TYPE "udt_API_Login"
VERSION : 0.1
   STRUCT
      Username : String[128];   // Username as entered in the login window / Request
      Password : String[128];   // User password as entered in the login window / Request
      AutoLogoffTime : Int;   // Minutes after the client must perform the logout if the user is idle.  / Response
      UserGroup : String[128];   // Name of the user group that the user belongs to. / Response
      LoginTriggerAndResponse : Int;   // 0 = ready/idle; 1 = request; 2 = OK (Login successful); 10 = UserNotFound; 11 = WrongPassword; 12 = Disabled; 13 = Locked; 14 = PasswordChangeRequired; 15 = PasswordChangeRequiredDomainUser / TriggerAndResponse
   END_STRUCT;

END_TYPE

TYPE "udt_API_Logout"
VERSION : 0.1
   STRUCT
      LogoutTriggerAndResponse : Int;   // 0 = ready/idle; 1 = request; 2 = OK (logout successful) / TriggerAndResponse
   END_STRUCT;

END_TYPE

TYPE "udt_API_Authorization"
VERSION : 0.1
   STRUCT
      AccessRightCustomId : String[20];   // Custom Id of the access right that the authorization is carried out against. / Request
      AuthorizationTriggerAndResponse : Int;   // 0 = ready/idle; 1 = request; 2 = OK (Authorized); 3 = OK (NotAuthorized); 4 = OK (Challenged): 12 = NoUserIsLoggedIn; 13 = AccessRightNotFound / TriggerAndResponse
      ElectronicSignatureType : Int;   // 0 = cleared; 1 = Confirmation only, optional comment; 2 = Confirmation only, required comment; 3 = Authenticated signature, optional comment; 4 = Authenticated signature, required comment / Response (optional)
      ElectronicSignatureName : String[128];   // Name of the required electronic signature / Response (optional)
      ElectronicSignatureUsername : String[128];   // Username to sign the electronic signature / Request (optional)
      ElectronicSignaturePassword : String[128];   // Password to sign the electronic signature / Request (optional)
      ElecronicSignatureComment : String[128];   // Comment provided with signing of the signature / Request (optional)
      ElectronicSignatureChallengeStatus : Int;   // 0 = cleared; 2 = OK; 10 = SignatoryAuthenticationError; 11 = SignatoryNotAuthorized; 12 = CommentRequired / Response (optional)
   END_STRUCT;

END_TYPE

TYPE "udt_API_UserDefinedEvent"
VERSION : 0.1
   STRUCT
      EventCustomId : String[20];   // Custom Id of the user defined event that is logged to the audit trail. / Request
      EventData : String[200];   // Data associated with the event (string separated with #).  / Request
      UserDefinedEventTriggerAndResponse : Int;   // 0 = ready/idle; 1 = request; 2 = OK (Event successfully written); 10 = EventCustomIdNotFound; 11 = EventDataNotConsistentWithEventTemplate / TriggerAndResponse
   END_STRUCT;

END_TYPE

TYPE "udt_API_StepRecipeDownload"
VERSION : 0.1
   STRUCT
      RecipeId : DInt;   // Id of selected recipe / Request
      StepNumber : DInt;   // Step number of the operation to be downloaded. First step starts with 1 / Request
      OperationId : DInt;   // Id of the operation that must be executed for the current procedural element.  / Response
      CreatedFromProceduralElement : DInt;   // Id of the procedural element, which is used to display the report data on the report. API writes the id of the procedural element from the recipe.  / Response
      StepRecipeDownloadTriggerAndResponse : Int;   // 0 = ready/idle; 1 = request; 2 = OK (step downloaded); 3 = OK (end of recipe); 10 = RecipeIdNotFound; 11 = ParameterAddressNotFoundOnServer; 12 = NonLinearRecipe; 13 = RecipeContainsNoSteps; 14 = NegativeOrZeroStepNumber; 15 = RecipeDoesNotHaveStepNumber / TriggerAndResponse
   END_STRUCT;

END_TYPE

TYPE "udt_API_TimeSync"
VERSION : 0.1
   STRUCT
      TimeSyncTriggerAndResponse : Int;   // 0 = ready/idle; 1 = request; 2 = OK (Time data sent) / TriggerAndResponse
      CurrentUnixServerTime : DInt;   // UNIX timestamp (seconds since Jan 01, 1970. (UTC)) / Response
      CurrentLocalServerTime : Date_And_Time;   // Current local server time in date time format. / Response
      CurrentUtcServerTime : Date_And_Time;   // Current UTC server time in date time format. / Response
      CurrentServerTimeOffset : Int;   // Number of hours representing the time offset from UTC / Response
   END_STRUCT;

END_TYPE

TYPE "udt_API_Watchdog"
VERSION : 0.1
   STRUCT
      IsApiResponsive : Bool;   // Periodically set to true by the API. Client should reset to false before checking the status of the service.  / Response
   END_STRUCT;

END_TYPE

TYPE "udt_API_ReportHeaderCreate"
VERSION : 0.1
   STRUCT
      StartUser : String[128];   // Name of the user that executed actions resulting in the generation of the report. / Request
      RecipeId : DInt;   // Id of the recipe that was executed to generate the report (in recipe regime only). Leave value at 0 for non-recipe regime. / Request (Optional)
      BatchId : DInt;   // Id of the batch that was executed to generate the report (in recipe regime only, if batches are used). Leave value at 0 if batch is not used. / Response
      ReportHeaderId : DInt;   // Id of the created report header. / Response
      ReportHeaderCreateTriggerAndResponse : Int;   // 0 = ready/idle; 1 = request; 2 = OK (Report header created); 10 = RecipeIdNotFound; 11 = BatchIdNotFound; 12 = RecipeIsNotLocalRecipe / TriggerAndResponse
   END_STRUCT;

END_TYPE

TYPE "udt_API_ReportStepUpload"
VERSION : 0.1
   STRUCT
      ReportHeaderId : DInt;   // Id of the report header to which the procedural element will be added. / Request
      OperationId : DInt;   // Id of the operation whose parameters are uploaded to the database. / Request
      StartDate : Date_And_Time;   // Start date and time of the procedural element / Request
      EndDate : Date_And_Time;   // End date and time of the procedural element / Request
      ExecutionStatus : Int;   // 0 = successful; 1 = failed; 2 = aborted / Request
      CreatedFromProceduralElement : DInt;   // Id of the procedural element from which the report data is created / Request (optional)
      ReportStepUploadTriggerAndResponse : Int;   // 0 = ready/idle; 1 = request; 2 = OK (Report step uploaded); 10 = ReportHeaderIdNotFound; 11 = OperationIdNotFound; 12 = InvalidExecutionStatus; 13 = ParameterAddressNotFoundOnServer; 14 = StartDateAfterEndDate / TriggerAndResponse
   END_STRUCT;

END_TYPE

TYPE "udt_API_ReportFinish"
VERSION : 0.1
   STRUCT
      EndUser : String[128];   // Name of the user that executed actions resulting in the completion of the report.
      ReportHeaderId : DInt;   // Id of the report header to be concluded
      ReportFinishTriggerAndResponse : Int;   // 0 = ready/idle, 1 = request, 2 = OK (Report header concluded), 10 = ReportHeaderIdNotFound
   END_STRUCT;

END_TYPE

TYPE "udt_API_Full"
VERSION : 0.1
   STRUCT
      Login : "udt_API_Login";
      Logout : "udt_API_Logout";
      Authorization : "udt_API_Authorization";
      UserDefinedEvent : "udt_API_UserDefinedEvent";
      StepRecipeDownload : "udt_API_StepRecipeDownload";
      TimeSync : "udt_API_TimeSync";
      Watchdog : "udt_API_Watchdog";
      ReportHeaderCreate : "udt_API_ReportHeaderCreate";
      ReportStepUpload : "udt_API_ReportStepUpload";
      ReportFinish : "udt_API_ReportFinish";
   END_STRUCT;

END_TYPE

TYPE "udtUnit"
VERSION : 0.1
   STRUCT
      Regime : Int;   //  Control mode (0=automatic, 1=manual, 2=service)
      Status : Int;   //  Unit status
      ID : Int;   //  Unit ID
      Ready : Int;   //  0 = Ready; 1 = not ready
      Enable : Bool;   //  1-Unit is Enabled
      Alocated : Bool;   //  1-Unit is alocated
      Spare1 : Bool;   // spare
      Active : Bool;   //  1-Unit is active
      AlarmAck : Bool;   //  1 = Akcknowledge all unit alarms
      interaction : Bool;   //  1 = unit request for operator interaction
      PhaseH : Bool;   //  1 = one or more phases are HELD
      PhaseF : Bool;   //  1 = one or more phases are in alarm
      Simulation : Bool;   // Enable Simulation on SCADA (ifix)
      Spare2 : Bool;   // Enable Simulation on HMI (siemens panel)
      Spare3 : Bool;   // spare
      Spare4 : Bool;
      Spare5 : Bool;
      Spare6 : Bool;
      Spare7 : Bool;
      Spare8 : Bool;
   END_STRUCT;

END_TYPE

DATA_BLOCK "dbAPI"
{ S7_Optimized_Access := 'FALSE' }
VERSION : 0.1
NON_RETAIN
   STRUCT
      PdbmApi : Array[0..4] of "udt_API_Full";
   END_STRUCT;


BEGIN
   PdbmApi[0].Login.Username := '';
   PdbmApi[0].Login.Password := '';
   PdbmApi[0].Login.AutoLogoffTime := 0;
   PdbmApi[0].Login.UserGroup := '';
   PdbmApi[0].Login.LoginTriggerAndResponse := 0;
   PdbmApi[0].Logout.LogoutTriggerAndResponse := 0;
   PdbmApi[0].Authorization.AccessRightCustomId := '';
   PdbmApi[0].Authorization.AuthorizationTriggerAndResponse := 0;
   PdbmApi[0].Authorization.ElectronicSignatureType := 0;
   PdbmApi[0].Authorization.ElectronicSignatureName := '';
   PdbmApi[0].Authorization.ElectronicSignatureUsername := '';
   PdbmApi[0].Authorization.ElectronicSignaturePassword := '';
   PdbmApi[0].Authorization.ElecronicSignatureComment := '';
   PdbmApi[0].Authorization.ElectronicSignatureChallengeStatus := 0;
   PdbmApi[0].UserDefinedEvent.EventCustomId := '';
   PdbmApi[0].UserDefinedEvent.EventData := '';
   PdbmApi[0].UserDefinedEvent.UserDefinedEventTriggerAndResponse := 2;
   PdbmApi[0].StepRecipeDownload.RecipeId := 0;
   PdbmApi[0].StepRecipeDownload.StepNumber := 0;
   PdbmApi[0].StepRecipeDownload.OperationId := 95;
   PdbmApi[0].StepRecipeDownload.CreatedFromProceduralElement := 157;
   PdbmApi[0].StepRecipeDownload.StepRecipeDownloadTriggerAndResponse := 0;
   PdbmApi[0].TimeSync.TimeSyncTriggerAndResponse := 0;
   PdbmApi[0].TimeSync.CurrentUnixServerTime := 1_671_231_209;
   PdbmApi[0].TimeSync.CurrentLocalServerTime := DT#2022-12-17-00:53:29.655;
   PdbmApi[0].TimeSync.CurrentUtcServerTime := DT#2022-12-16-22:53:29.656;
   PdbmApi[0].TimeSync.CurrentServerTimeOffset := 2;
   PdbmApi[0].Watchdog.IsApiResponsive := FALSE;
   PdbmApi[0].ReportHeaderCreate.StartUser := '';
   PdbmApi[0].ReportHeaderCreate.RecipeId := 0;
   PdbmApi[0].ReportHeaderCreate.BatchId := 0;
   PdbmApi[0].ReportHeaderCreate.ReportHeaderId := 1491;
   PdbmApi[0].ReportHeaderCreate.ReportHeaderCreateTriggerAndResponse := 0;
   PdbmApi[0].ReportStepUpload.ReportHeaderId := 0;
   PdbmApi[0].ReportStepUpload.OperationId := 0;
   PdbmApi[0].ReportStepUpload.StartDate := DT#1990-01-01-00:00:00;
   PdbmApi[0].ReportStepUpload.EndDate := DT#1990-01-01-00:00:00;
   PdbmApi[0].ReportStepUpload.ExecutionStatus := 0;
   PdbmApi[0].ReportStepUpload.CreatedFromProceduralElement := 0;
   PdbmApi[0].ReportStepUpload.ReportStepUploadTriggerAndResponse := 0;
   PdbmApi[0].ReportFinish.EndUser := '';
   PdbmApi[0].ReportFinish.ReportHeaderId := 0;
   PdbmApi[0].ReportFinish.ReportFinishTriggerAndResponse := 2;
   PdbmApi[1].Login.Username := '';
   PdbmApi[1].Login.Password := '';
   PdbmApi[1].Login.AutoLogoffTime := 60;
   PdbmApi[1].Login.UserGroup := 'ADMINISTRATOR';
   PdbmApi[1].Login.LoginTriggerAndResponse := 0;
   PdbmApi[1].Logout.LogoutTriggerAndResponse := 2;
   PdbmApi[1].Authorization.AccessRightCustomId := '';
   PdbmApi[1].Authorization.AuthorizationTriggerAndResponse := 0;
   PdbmApi[1].Authorization.ElectronicSignatureType := 0;
   PdbmApi[1].Authorization.ElectronicSignatureName := '';
   PdbmApi[1].Authorization.ElectronicSignatureUsername := '';
   PdbmApi[1].Authorization.ElectronicSignaturePassword := '';
   PdbmApi[1].Authorization.ElecronicSignatureComment := '';
   PdbmApi[1].Authorization.ElectronicSignatureChallengeStatus := 0;
   PdbmApi[1].UserDefinedEvent.EventCustomId := '';
   PdbmApi[1].UserDefinedEvent.EventData := '';
   PdbmApi[1].UserDefinedEvent.UserDefinedEventTriggerAndResponse := 2;
   PdbmApi[1].StepRecipeDownload.RecipeId := 0;
   PdbmApi[1].StepRecipeDownload.StepNumber := 0;
   PdbmApi[1].StepRecipeDownload.OperationId := 0;
   PdbmApi[1].StepRecipeDownload.CreatedFromProceduralElement := 0;
   PdbmApi[1].StepRecipeDownload.StepRecipeDownloadTriggerAndResponse := 0;
   PdbmApi[1].TimeSync.TimeSyncTriggerAndResponse := 0;
   PdbmApi[1].TimeSync.CurrentUnixServerTime := 0;
   PdbmApi[1].TimeSync.CurrentLocalServerTime := DT#1990-01-01-00:00:00;
   PdbmApi[1].TimeSync.CurrentUtcServerTime := DT#1990-01-01-00:00:00;
   PdbmApi[1].TimeSync.CurrentServerTimeOffset := 0;
   PdbmApi[1].Watchdog.IsApiResponsive := TRUE;
   PdbmApi[1].ReportHeaderCreate.StartUser := '';
   PdbmApi[1].ReportHeaderCreate.RecipeId := 0;
   PdbmApi[1].ReportHeaderCreate.BatchId := 0;
   PdbmApi[1].ReportHeaderCreate.ReportHeaderId := 0;
   PdbmApi[1].ReportHeaderCreate.ReportHeaderCreateTriggerAndResponse := 0;
   PdbmApi[1].ReportStepUpload.ReportHeaderId := 0;
   PdbmApi[1].ReportStepUpload.OperationId := 0;
   PdbmApi[1].ReportStepUpload.StartDate := DT#1990-01-01-00:00:00;
   PdbmApi[1].ReportStepUpload.EndDate := DT#1990-01-01-00:00:00;
   PdbmApi[1].ReportStepUpload.ExecutionStatus := 0;
   PdbmApi[1].ReportStepUpload.CreatedFromProceduralElement := 0;
   PdbmApi[1].ReportStepUpload.ReportStepUploadTriggerAndResponse := 0;
   PdbmApi[1].ReportFinish.EndUser := '';
   PdbmApi[1].ReportFinish.ReportHeaderId := 0;
   PdbmApi[1].ReportFinish.ReportFinishTriggerAndResponse := 0;
   PdbmApi[2].Login.Username := '';
   PdbmApi[2].Login.Password := '';
   PdbmApi[2].Login.AutoLogoffTime := 60;
   PdbmApi[2].Login.UserGroup := 'ADMINISTRATOR';
   PdbmApi[2].Login.LoginTriggerAndResponse := 0;
   PdbmApi[2].Logout.LogoutTriggerAndResponse := 2;
   PdbmApi[2].Authorization.AccessRightCustomId := '0';
   PdbmApi[2].Authorization.AuthorizationTriggerAndResponse := 0;
   PdbmApi[2].Authorization.ElectronicSignatureType := 0;
   PdbmApi[2].Authorization.ElectronicSignatureName := '';
   PdbmApi[2].Authorization.ElectronicSignatureUsername := '';
   PdbmApi[2].Authorization.ElectronicSignaturePassword := '';
   PdbmApi[2].Authorization.ElecronicSignatureComment := '';
   PdbmApi[2].Authorization.ElectronicSignatureChallengeStatus := 0;
   PdbmApi[2].UserDefinedEvent.EventCustomId := '';
   PdbmApi[2].UserDefinedEvent.EventData := '';
   PdbmApi[2].UserDefinedEvent.UserDefinedEventTriggerAndResponse := 2;
   PdbmApi[2].StepRecipeDownload.RecipeId := 0;
   PdbmApi[2].StepRecipeDownload.StepNumber := 0;
   PdbmApi[2].StepRecipeDownload.OperationId := 0;
   PdbmApi[2].StepRecipeDownload.CreatedFromProceduralElement := 0;
   PdbmApi[2].StepRecipeDownload.StepRecipeDownloadTriggerAndResponse := 0;
   PdbmApi[2].TimeSync.TimeSyncTriggerAndResponse := 0;
   PdbmApi[2].TimeSync.CurrentUnixServerTime := 0;
   PdbmApi[2].TimeSync.CurrentLocalServerTime := DT#1990-01-01-00:00:00;
   PdbmApi[2].TimeSync.CurrentUtcServerTime := DT#1990-01-01-00:00:00;
   PdbmApi[2].TimeSync.CurrentServerTimeOffset := 0;
   PdbmApi[2].Watchdog.IsApiResponsive := TRUE;
   PdbmApi[2].ReportHeaderCreate.StartUser := '';
   PdbmApi[2].ReportHeaderCreate.RecipeId := 0;
   PdbmApi[2].ReportHeaderCreate.BatchId := 0;
   PdbmApi[2].ReportHeaderCreate.ReportHeaderId := 0;
   PdbmApi[2].ReportHeaderCreate.ReportHeaderCreateTriggerAndResponse := 0;
   PdbmApi[2].ReportStepUpload.ReportHeaderId := 0;
   PdbmApi[2].ReportStepUpload.OperationId := 0;
   PdbmApi[2].ReportStepUpload.StartDate := DT#1990-01-01-00:00:00;
   PdbmApi[2].ReportStepUpload.EndDate := DT#1990-01-01-00:00:00;
   PdbmApi[2].ReportStepUpload.ExecutionStatus := 0;
   PdbmApi[2].ReportStepUpload.CreatedFromProceduralElement := 0;
   PdbmApi[2].ReportStepUpload.ReportStepUploadTriggerAndResponse := 0;
   PdbmApi[2].ReportFinish.EndUser := '';
   PdbmApi[2].ReportFinish.ReportHeaderId := 0;
   PdbmApi[2].ReportFinish.ReportFinishTriggerAndResponse := 0;
   PdbmApi[3].Login.Username := '';
   PdbmApi[3].Login.Password := '';
   PdbmApi[3].Login.AutoLogoffTime := 60;
   PdbmApi[3].Login.UserGroup := 'ADMINISTRATOR';
   PdbmApi[3].Login.LoginTriggerAndResponse := 0;
   PdbmApi[3].Logout.LogoutTriggerAndResponse := 2;
   PdbmApi[3].Authorization.AccessRightCustomId := '';
   PdbmApi[3].Authorization.AuthorizationTriggerAndResponse := 0;
   PdbmApi[3].Authorization.ElectronicSignatureType := 0;
   PdbmApi[3].Authorization.ElectronicSignatureName := '';
   PdbmApi[3].Authorization.ElectronicSignatureUsername := '';
   PdbmApi[3].Authorization.ElectronicSignaturePassword := '';
   PdbmApi[3].Authorization.ElecronicSignatureComment := '';
   PdbmApi[3].Authorization.ElectronicSignatureChallengeStatus := 0;
   PdbmApi[3].UserDefinedEvent.EventCustomId := '';
   PdbmApi[3].UserDefinedEvent.EventData := '';
   PdbmApi[3].UserDefinedEvent.UserDefinedEventTriggerAndResponse := 2;
   PdbmApi[3].StepRecipeDownload.RecipeId := 0;
   PdbmApi[3].StepRecipeDownload.StepNumber := 0;
   PdbmApi[3].StepRecipeDownload.OperationId := 0;
   PdbmApi[3].StepRecipeDownload.CreatedFromProceduralElement := 0;
   PdbmApi[3].StepRecipeDownload.StepRecipeDownloadTriggerAndResponse := 0;
   PdbmApi[3].TimeSync.TimeSyncTriggerAndResponse := 0;
   PdbmApi[3].TimeSync.CurrentUnixServerTime := 0;
   PdbmApi[3].TimeSync.CurrentLocalServerTime := DT#1990-01-01-00:00:00;
   PdbmApi[3].TimeSync.CurrentUtcServerTime := DT#1990-01-01-00:00:00;
   PdbmApi[3].TimeSync.CurrentServerTimeOffset := 0;
   PdbmApi[3].Watchdog.IsApiResponsive := TRUE;
   PdbmApi[3].ReportHeaderCreate.StartUser := '';
   PdbmApi[3].ReportHeaderCreate.RecipeId := 0;
   PdbmApi[3].ReportHeaderCreate.BatchId := 0;
   PdbmApi[3].ReportHeaderCreate.ReportHeaderId := 0;
   PdbmApi[3].ReportHeaderCreate.ReportHeaderCreateTriggerAndResponse := 0;
   PdbmApi[3].ReportStepUpload.ReportHeaderId := 0;
   PdbmApi[3].ReportStepUpload.OperationId := 0;
   PdbmApi[3].ReportStepUpload.StartDate := DT#1990-01-01-00:00:00;
   PdbmApi[3].ReportStepUpload.EndDate := DT#1990-01-01-00:00:00;
   PdbmApi[3].ReportStepUpload.ExecutionStatus := 0;
   PdbmApi[3].ReportStepUpload.CreatedFromProceduralElement := 0;
   PdbmApi[3].ReportStepUpload.ReportStepUploadTriggerAndResponse := 0;
   PdbmApi[3].ReportFinish.EndUser := '';
   PdbmApi[3].ReportFinish.ReportHeaderId := 0;
   PdbmApi[3].ReportFinish.ReportFinishTriggerAndResponse := 0;
   PdbmApi[4].Login.Username := '';
   PdbmApi[4].Login.Password := '';
   PdbmApi[4].Login.AutoLogoffTime := 0;
   PdbmApi[4].Login.UserGroup := '';
   PdbmApi[4].Login.LoginTriggerAndResponse := 0;
   PdbmApi[4].Logout.LogoutTriggerAndResponse := 0;
   PdbmApi[4].Authorization.AccessRightCustomId := '';
   PdbmApi[4].Authorization.AuthorizationTriggerAndResponse := 0;
   PdbmApi[4].Authorization.ElectronicSignatureType := 0;
   PdbmApi[4].Authorization.ElectronicSignatureName := '';
   PdbmApi[4].Authorization.ElectronicSignatureUsername := '';
   PdbmApi[4].Authorization.ElectronicSignaturePassword := '';
   PdbmApi[4].Authorization.ElecronicSignatureComment := '';
   PdbmApi[4].Authorization.ElectronicSignatureChallengeStatus := 0;
   PdbmApi[4].UserDefinedEvent.EventCustomId := '';
   PdbmApi[4].UserDefinedEvent.EventData := '';
   PdbmApi[4].UserDefinedEvent.UserDefinedEventTriggerAndResponse := 0;
   PdbmApi[4].StepRecipeDownload.RecipeId := 0;
   PdbmApi[4].StepRecipeDownload.StepNumber := 0;
   PdbmApi[4].StepRecipeDownload.OperationId := 0;
   PdbmApi[4].StepRecipeDownload.CreatedFromProceduralElement := 0;
   PdbmApi[4].StepRecipeDownload.StepRecipeDownloadTriggerAndResponse := 0;
   PdbmApi[4].TimeSync.TimeSyncTriggerAndResponse := 0;
   PdbmApi[4].TimeSync.CurrentUnixServerTime := 0;
   PdbmApi[4].TimeSync.CurrentLocalServerTime := DT#1990-01-01-00:00:00;
   PdbmApi[4].TimeSync.CurrentUtcServerTime := DT#1990-01-01-00:00:00;
   PdbmApi[4].TimeSync.CurrentServerTimeOffset := 0;
   PdbmApi[4].Watchdog.IsApiResponsive := TRUE;
   PdbmApi[4].ReportHeaderCreate.StartUser := '';
   PdbmApi[4].ReportHeaderCreate.RecipeId := 0;
   PdbmApi[4].ReportHeaderCreate.BatchId := 0;
   PdbmApi[4].ReportHeaderCreate.ReportHeaderId := 145;
   PdbmApi[4].ReportHeaderCreate.ReportHeaderCreateTriggerAndResponse := 2;
   PdbmApi[4].ReportStepUpload.ReportHeaderId := 0;
   PdbmApi[4].ReportStepUpload.OperationId := 0;
   PdbmApi[4].ReportStepUpload.StartDate := DT#1990-01-01-00:00:00;
   PdbmApi[4].ReportStepUpload.EndDate := DT#1990-01-01-00:00:00;
   PdbmApi[4].ReportStepUpload.ExecutionStatus := 0;
   PdbmApi[4].ReportStepUpload.CreatedFromProceduralElement := 0;
   PdbmApi[4].ReportStepUpload.ReportStepUploadTriggerAndResponse := 2;
   PdbmApi[4].ReportFinish.EndUser := '';
   PdbmApi[4].ReportFinish.ReportHeaderId := 0;
   PdbmApi[4].ReportFinish.ReportFinishTriggerAndResponse := 0;

END_DATA_BLOCK

DATA_BLOCK "dbUnit"
{ S7_Optimized_Access := 'FALSE' }
VERSION : 0.1
   STRUCT
      Unit : Array[1..10] of "udtUnit";
   END_STRUCT;


BEGIN
   Unit[1].Regime := 0;
   Unit[1].Status := 2;
   Unit[1].ID := 1;
   Unit[1].Ready := 0;
   Unit[1].Enable := TRUE;
   Unit[1].Alocated := FALSE;
   Unit[1].Spare1 := FALSE;
   Unit[1].Active := TRUE;
   Unit[1].AlarmAck := FALSE;
   Unit[1].interaction := FALSE;
   Unit[1].PhaseH := TRUE;
   Unit[1].PhaseF := FALSE;
   Unit[1].Simulation := TRUE;
   Unit[1].Spare2 := FALSE;
   Unit[1].Spare3 := FALSE;
   Unit[1].Spare4 := FALSE;
   Unit[1].Spare5 := FALSE;
   Unit[1].Spare6 := FALSE;
   Unit[1].Spare7 := FALSE;
   Unit[1].Spare8 := FALSE;
   Unit[2].Regime := 0;
   Unit[2].Status := 2;
   Unit[2].ID := 2;
   Unit[2].Ready := 0;
   Unit[2].Enable := TRUE;
   Unit[2].Alocated := FALSE;
   Unit[2].Spare1 := FALSE;
   Unit[2].Active := TRUE;
   Unit[2].AlarmAck := TRUE;
   Unit[2].interaction := FALSE;
   Unit[2].PhaseH := TRUE;
   Unit[2].PhaseF := FALSE;
   Unit[2].Simulation := FALSE;
   Unit[2].Spare2 := FALSE;
   Unit[2].Spare3 := FALSE;
   Unit[2].Spare4 := FALSE;
   Unit[2].Spare5 := FALSE;
   Unit[2].Spare6 := FALSE;
   Unit[2].Spare7 := FALSE;
   Unit[2].Spare8 := FALSE;
   Unit[3].Regime := 0;
   Unit[3].Status := 2;
   Unit[3].ID := 3;
   Unit[3].Ready := 0;
   Unit[3].Enable := TRUE;
   Unit[3].Alocated := FALSE;
   Unit[3].Spare1 := FALSE;
   Unit[3].Active := TRUE;
   Unit[3].AlarmAck := TRUE;
   Unit[3].interaction := TRUE;
   Unit[3].PhaseH := FALSE;
   Unit[3].PhaseF := FALSE;
   Unit[3].Simulation := FALSE;
   Unit[3].Spare2 := FALSE;
   Unit[3].Spare3 := FALSE;
   Unit[3].Spare4 := FALSE;
   Unit[3].Spare5 := FALSE;
   Unit[3].Spare6 := FALSE;
   Unit[3].Spare7 := FALSE;
   Unit[3].Spare8 := FALSE;
   Unit[4].Regime := 0;
   Unit[4].Status := 2;
   Unit[4].ID := 4;
   Unit[4].Ready := 0;
   Unit[4].Enable := TRUE;
   Unit[4].Alocated := FALSE;
   Unit[4].Spare1 := FALSE;
   Unit[4].Active := TRUE;
   Unit[4].AlarmAck := TRUE;
   Unit[4].interaction := FALSE;
   Unit[4].PhaseH := TRUE;
   Unit[4].PhaseF := FALSE;
   Unit[4].Simulation := FALSE;
   Unit[4].Spare2 := FALSE;
   Unit[4].Spare3 := FALSE;
   Unit[4].Spare4 := FALSE;
   Unit[4].Spare5 := FALSE;
   Unit[4].Spare6 := FALSE;
   Unit[4].Spare7 := FALSE;
   Unit[4].Spare8 := FALSE;
   Unit[5].Regime := 0;
   Unit[5].Status := 2;
   Unit[5].ID := 5;
   Unit[5].Ready := 0;
   Unit[5].Enable := TRUE;
   Unit[5].Alocated := FALSE;
   Unit[5].Spare1 := FALSE;
   Unit[5].Active := TRUE;
   Unit[5].AlarmAck := TRUE;
   Unit[5].interaction := FALSE;
   Unit[5].PhaseH := TRUE;
   Unit[5].PhaseF := FALSE;
   Unit[5].Simulation := FALSE;
   Unit[5].Spare2 := FALSE;
   Unit[5].Spare3 := FALSE;
   Unit[5].Spare4 := FALSE;
   Unit[5].Spare5 := FALSE;
   Unit[5].Spare6 := FALSE;
   Unit[5].Spare7 := FALSE;
   Unit[5].Spare8 := FALSE;
   Unit[6].Regime := 0;
   Unit[6].Status := 1;
   Unit[6].ID := 6;
   Unit[6].Ready := 0;
   Unit[6].Enable := TRUE;
   Unit[6].Alocated := FALSE;
   Unit[6].Spare1 := FALSE;
   Unit[6].Active := FALSE;
   Unit[6].AlarmAck := TRUE;
   Unit[6].interaction := FALSE;
   Unit[6].PhaseH := FALSE;
   Unit[6].PhaseF := FALSE;
   Unit[6].Simulation := FALSE;
   Unit[6].Spare2 := FALSE;
   Unit[6].Spare3 := FALSE;
   Unit[6].Spare4 := FALSE;
   Unit[6].Spare5 := FALSE;
   Unit[6].Spare6 := FALSE;
   Unit[6].Spare7 := FALSE;
   Unit[6].Spare8 := FALSE;
   Unit[7].Regime := 0;
   Unit[7].Status := 1;
   Unit[7].ID := 7;
   Unit[7].Ready := 0;
   Unit[7].Enable := TRUE;
   Unit[7].Alocated := FALSE;
   Unit[7].Spare1 := FALSE;
   Unit[7].Active := FALSE;
   Unit[7].AlarmAck := TRUE;
   Unit[7].interaction := FALSE;
   Unit[7].PhaseH := FALSE;
   Unit[7].PhaseF := FALSE;
   Unit[7].Simulation := FALSE;
   Unit[7].Spare2 := FALSE;
   Unit[7].Spare3 := FALSE;
   Unit[7].Spare4 := FALSE;
   Unit[7].Spare5 := FALSE;
   Unit[7].Spare6 := FALSE;
   Unit[7].Spare7 := FALSE;
   Unit[7].Spare8 := FALSE;
   Unit[8].Regime := 0;
   Unit[8].Status := 1;
   Unit[8].ID := 8;
   Unit[8].Ready := 0;
   Unit[8].Enable := TRUE;
   Unit[8].Alocated := FALSE;
   Unit[8].Spare1 := FALSE;
   Unit[8].Active := FALSE;
   Unit[8].AlarmAck := TRUE;
   Unit[8].interaction := FALSE;
   Unit[8].PhaseH := FALSE;
   Unit[8].PhaseF := FALSE;
   Unit[8].Simulation := FALSE;
   Unit[8].Spare2 := FALSE;
   Unit[8].Spare3 := FALSE;
   Unit[8].Spare4 := FALSE;
   Unit[8].Spare5 := FALSE;
   Unit[8].Spare6 := FALSE;
   Unit[8].Spare7 := FALSE;
   Unit[8].Spare8 := FALSE;
   Unit[9].Regime := 0;
   Unit[9].Status := 0;
   Unit[9].ID := 9;
   Unit[9].Ready := 0;
   Unit[9].Enable := TRUE;
   Unit[9].Alocated := FALSE;
   Unit[9].Spare1 := FALSE;
   Unit[9].Active := FALSE;
   Unit[9].AlarmAck := TRUE;
   Unit[9].interaction := FALSE;
   Unit[9].PhaseH := FALSE;
   Unit[9].PhaseF := FALSE;
   Unit[9].Simulation := FALSE;
   Unit[9].Spare2 := FALSE;
   Unit[9].Spare3 := FALSE;
   Unit[9].Spare4 := FALSE;
   Unit[9].Spare5 := FALSE;
   Unit[9].Spare6 := FALSE;
   Unit[9].Spare7 := FALSE;
   Unit[9].Spare8 := FALSE;
   Unit[10].Regime := 0;
   Unit[10].Status := 0;
   Unit[10].ID := 10;
   Unit[10].Ready := 0;
   Unit[10].Enable := TRUE;
   Unit[10].Alocated := FALSE;
   Unit[10].Spare1 := FALSE;
   Unit[10].Active := FALSE;
   Unit[10].AlarmAck := TRUE;
   Unit[10].interaction := FALSE;
   Unit[10].PhaseH := FALSE;
   Unit[10].PhaseF := FALSE;
   Unit[10].Simulation := FALSE;
   Unit[10].Spare2 := FALSE;
   Unit[10].Spare3 := FALSE;
   Unit[10].Spare4 := FALSE;
   Unit[10].Spare5 := FALSE;
   Unit[10].Spare6 := FALSE;
   Unit[10].Spare7 := FALSE;
   Unit[10].Spare8 := FALSE;

END_DATA_BLOCK

DATA_BLOCK "dbPLI"
{ S7_Optimized_Access := 'FALSE' }
VERSION : 1.0
   STRUCT
      PLI_EX : Array[1..150] of Int;
      PLI_ST : Array[1..150] of Int;
      PLI_SI : Array[1..150] of Int;
      PLI_OP : Array[1..150] of Int;
      PLI_WR : Array[1..150] of Word;
      PLI_OC : Array[1..150] of Int;
      PLI_CD : Array[1..150] of Int;
      PLI_IS : Array[1..150] of Int;
      PLI_UN : Array[1..150] of Int;
      PLI_F : Array[1..150] of Int;
      PLI_RQ : Array[1..150] of Int;
      PLI_SB : Array[1..150] of Int;
      PLI_BRQ : Array[1..150] of Int;
      PLI_HI : Array[1..150] of Int;
      PLI_MS : Array[1..150] of Int;
      PLI_MD : Array[1..150] of Int;
      PLI_RC : Array[1..150] of Bool;
      PLI_TC : Array[1..150] of Bool;
      PLI_AC : Array[1..150] of Bool;
      PLI_HC : Array[1..150] of Bool;
      PLI_SC : Array[1..150] of Bool;
      PLI_EC : Array[1..150] of Bool;
      PLI_R : Array[1..150] of Bool;
      PLI_T : Array[1..150] of Bool;
      PLI_A : Array[1..150] of Bool;
      PLI_H : Array[1..150] of Bool;
      PLI_S : Array[1..150] of Bool;
      PLI_E : Array[1..150] of Bool;
      PLI_I : Array[1..150] of Bool;
      PLI_C : Array[1..150] of Bool;
      PLI_AD : Array[1..150] of Bool;
      PLI_HD : Array[1..150] of Bool;
      PLI_SD : Array[1..150] of Bool;
      PLI_FI : Array[1..150] of Bool;
      PLI_W : Array[1..150] of Bool;
      PLI_P : Array[1..150] of Bool;
      PLI_PD : Array[1..150] of Bool;
      PLI_SS : Array[1..150] of Bool;
      PLI_NC : Array[1..150] of Bool;
      PLI_IN : Array[1..150] of Bool;
      PLI_ER : Array[1..150] of Bool;
      PLI_OR : Array[1..150] of Bool;
      PLI_RR : Array[1..150] of Bool;
      PLI_CR : Array[1..150] of Bool;
      PLI_RE : Array[1..150] of Bool;
      PLI_DL : Array[1..150] of Bool;
      PLI_WC : Array[1..150] of Bool;
      PLI_II : Array[1..150] of Bool;
      PLI_HA : Array[1..150] of Bool;
   END_STRUCT;


BEGIN
   PLI_EX[1] := 0;
   PLI_EX[2] := 0;
   PLI_EX[3] := 0;
   PLI_EX[4] := 0;
   PLI_EX[5] := 0;
   PLI_EX[6] := 0;
   PLI_EX[7] := 0;
   PLI_EX[8] := 0;
   PLI_EX[9] := 0;
   PLI_EX[10] := 0;
   PLI_EX[11] := 0;
   PLI_EX[12] := 0;
   PLI_EX[13] := 0;
   PLI_EX[14] := 0;
   PLI_EX[15] := 0;
   PLI_EX[16] := 0;
   PLI_EX[17] := 0;
   PLI_EX[18] := 0;
   PLI_EX[19] := 0;
   PLI_EX[20] := 0;
   PLI_EX[21] := 0;
   PLI_EX[22] := 0;
   PLI_EX[23] := 0;
   PLI_EX[24] := 0;
   PLI_EX[25] := 0;
   PLI_EX[26] := 0;
   PLI_EX[27] := 0;
   PLI_EX[28] := 0;
   PLI_EX[29] := 0;
   PLI_EX[30] := 0;
   PLI_EX[31] := 0;
   PLI_EX[32] := 0;
   PLI_EX[33] := 0;
   PLI_EX[34] := 0;
   PLI_EX[35] := 0;
   PLI_EX[36] := 0;
   PLI_EX[37] := 0;
   PLI_EX[38] := 0;
   PLI_EX[39] := 0;
   PLI_EX[40] := 0;
   PLI_EX[41] := 0;
   PLI_EX[42] := 0;
   PLI_EX[43] := 0;
   PLI_EX[44] := 0;
   PLI_EX[45] := 0;
   PLI_EX[46] := 0;
   PLI_EX[47] := 0;
   PLI_EX[48] := 0;
   PLI_EX[49] := 0;
   PLI_EX[50] := 0;
   PLI_EX[51] := 0;
   PLI_EX[52] := 0;
   PLI_EX[53] := 0;
   PLI_EX[54] := 0;
   PLI_EX[55] := 0;
   PLI_EX[56] := 0;
   PLI_EX[57] := 0;
   PLI_EX[58] := 0;
   PLI_EX[59] := 0;
   PLI_EX[60] := 0;
   PLI_EX[61] := 0;
   PLI_EX[62] := 0;
   PLI_EX[63] := 0;
   PLI_EX[64] := 0;
   PLI_EX[65] := 0;
   PLI_EX[66] := 0;
   PLI_EX[67] := 0;
   PLI_EX[68] := 0;
   PLI_EX[69] := 0;
   PLI_EX[70] := 0;
   PLI_EX[71] := 0;
   PLI_EX[72] := 0;
   PLI_EX[73] := 0;
   PLI_EX[74] := 0;
   PLI_EX[75] := 0;
   PLI_EX[76] := 0;
   PLI_EX[77] := 0;
   PLI_EX[78] := 0;
   PLI_EX[79] := 0;
   PLI_EX[80] := 0;
   PLI_EX[81] := 0;
   PLI_EX[82] := 0;
   PLI_EX[83] := 0;
   PLI_EX[84] := 0;
   PLI_EX[85] := 0;
   PLI_EX[86] := 0;
   PLI_EX[87] := 0;
   PLI_EX[88] := 0;
   PLI_EX[89] := 0;
   PLI_EX[90] := 0;
   PLI_EX[91] := 0;
   PLI_EX[92] := 0;
   PLI_EX[93] := 0;
   PLI_EX[94] := 0;
   PLI_EX[95] := 0;
   PLI_EX[96] := 0;
   PLI_EX[97] := 0;
   PLI_EX[98] := 0;
   PLI_EX[99] := 0;
   PLI_EX[100] := 0;
   PLI_EX[101] := 0;
   PLI_EX[102] := 0;
   PLI_EX[103] := 0;
   PLI_EX[104] := 0;
   PLI_EX[105] := 0;
   PLI_EX[106] := 0;
   PLI_EX[107] := 0;
   PLI_EX[108] := 0;
   PLI_EX[109] := 0;
   PLI_EX[110] := 0;
   PLI_EX[111] := 0;
   PLI_EX[112] := 0;
   PLI_EX[113] := 0;
   PLI_EX[114] := 0;
   PLI_EX[115] := 0;
   PLI_EX[116] := 0;
   PLI_EX[117] := 0;
   PLI_EX[118] := 0;
   PLI_EX[119] := 0;
   PLI_EX[120] := 0;
   PLI_EX[121] := 0;
   PLI_EX[122] := 0;
   PLI_EX[123] := 0;
   PLI_EX[124] := 0;
   PLI_EX[125] := 0;
   PLI_EX[126] := 0;
   PLI_EX[127] := 0;
   PLI_EX[128] := 0;
   PLI_EX[129] := 0;
   PLI_EX[130] := 0;
   PLI_EX[131] := 0;
   PLI_EX[132] := 0;
   PLI_EX[133] := 0;
   PLI_EX[134] := 0;
   PLI_EX[135] := 0;
   PLI_EX[136] := 0;
   PLI_EX[137] := 0;
   PLI_EX[138] := 0;
   PLI_EX[139] := 0;
   PLI_EX[140] := 0;
   PLI_EX[141] := 0;
   PLI_EX[142] := 0;
   PLI_EX[143] := 0;
   PLI_EX[144] := 0;
   PLI_EX[145] := 0;
   PLI_EX[146] := 0;
   PLI_EX[147] := 0;
   PLI_EX[148] := 0;
   PLI_EX[149] := 0;
   PLI_EX[150] := 0;
   PLI_ST[1] := 100;
   PLI_ST[2] := 100;
   PLI_ST[3] := 100;
   PLI_ST[4] := 100;
   PLI_ST[5] := 100;
   PLI_ST[6] := 100;
   PLI_ST[7] := 100;
   PLI_ST[8] := 100;
   PLI_ST[9] := 100;
   PLI_ST[10] := 100;
   PLI_ST[11] := 100;
   PLI_ST[12] := 100;
   PLI_ST[13] := 100;
   PLI_ST[14] := 100;
   PLI_ST[15] := 100;
   PLI_ST[16] := 100;
   PLI_ST[17] := 100;
   PLI_ST[18] := 100;
   PLI_ST[19] := 100;
   PLI_ST[20] := 100;
   PLI_ST[21] := 100;
   PLI_ST[22] := 100;
   PLI_ST[23] := 100;
   PLI_ST[24] := 100;
   PLI_ST[25] := 100;
   PLI_ST[26] := 100;
   PLI_ST[27] := 100;
   PLI_ST[28] := 100;
   PLI_ST[29] := 100;
   PLI_ST[30] := 100;
   PLI_ST[31] := 100;
   PLI_ST[32] := 100;
   PLI_ST[33] := 100;
   PLI_ST[34] := 100;
   PLI_ST[35] := 100;
   PLI_ST[36] := 100;
   PLI_ST[37] := 100;
   PLI_ST[38] := 100;
   PLI_ST[39] := 100;
   PLI_ST[40] := 100;
   PLI_ST[41] := 100;
   PLI_ST[42] := 100;
   PLI_ST[43] := 100;
   PLI_ST[44] := 100;
   PLI_ST[45] := 100;
   PLI_ST[46] := 100;
   PLI_ST[47] := 100;
   PLI_ST[48] := 100;
   PLI_ST[49] := 100;
   PLI_ST[50] := 100;
   PLI_ST[51] := 100;
   PLI_ST[52] := 100;
   PLI_ST[53] := 100;
   PLI_ST[54] := 100;
   PLI_ST[55] := 100;
   PLI_ST[56] := 100;
   PLI_ST[57] := 100;
   PLI_ST[58] := 100;
   PLI_ST[59] := 100;
   PLI_ST[60] := 100;
   PLI_ST[61] := 100;
   PLI_ST[62] := 100;
   PLI_ST[63] := 100;
   PLI_ST[64] := 100;
   PLI_ST[65] := 100;
   PLI_ST[66] := 100;
   PLI_ST[67] := 100;
   PLI_ST[68] := 100;
   PLI_ST[69] := 100;
   PLI_ST[70] := 100;
   PLI_ST[71] := 100;
   PLI_ST[72] := 100;
   PLI_ST[73] := 100;
   PLI_ST[74] := 100;
   PLI_ST[75] := 100;
   PLI_ST[76] := 100;
   PLI_ST[77] := 100;
   PLI_ST[78] := 100;
   PLI_ST[79] := 100;
   PLI_ST[80] := 100;
   PLI_ST[81] := 100;
   PLI_ST[82] := 100;
   PLI_ST[83] := 100;
   PLI_ST[84] := 100;
   PLI_ST[85] := 100;
   PLI_ST[86] := 100;
   PLI_ST[87] := 100;
   PLI_ST[88] := 100;
   PLI_ST[89] := 100;
   PLI_ST[90] := 100;
   PLI_ST[91] := 100;
   PLI_ST[92] := 100;
   PLI_ST[93] := 100;
   PLI_ST[94] := 100;
   PLI_ST[95] := 100;
   PLI_ST[96] := 100;
   PLI_ST[97] := 100;
   PLI_ST[98] := 100;
   PLI_ST[99] := 100;
   PLI_ST[100] := 100;
   PLI_ST[101] := 100;
   PLI_ST[102] := 100;
   PLI_ST[103] := 100;
   PLI_ST[104] := 100;
   PLI_ST[105] := 100;
   PLI_ST[106] := 100;
   PLI_ST[107] := 100;
   PLI_ST[108] := 100;
   PLI_ST[109] := 100;
   PLI_ST[110] := 50;
   PLI_ST[111] := 50;
   PLI_ST[112] := 20;
   PLI_ST[113] := 100;
   PLI_ST[114] := 100;
   PLI_ST[115] := 20;
   PLI_ST[116] := 50;
   PLI_ST[117] := 100;
   PLI_ST[118] := 100;
   PLI_ST[119] := 100;
   PLI_ST[120] := 100;
   PLI_ST[121] := 100;
   PLI_ST[122] := 100;
   PLI_ST[123] := 100;
   PLI_ST[124] := 100;
   PLI_ST[125] := 100;
   PLI_ST[126] := 100;
   PLI_ST[127] := 100;
   PLI_ST[128] := 100;
   PLI_ST[129] := 100;
   PLI_ST[130] := 100;
   PLI_ST[131] := 100;
   PLI_ST[132] := 100;
   PLI_ST[133] := 100;
   PLI_ST[134] := 100;
   PLI_ST[135] := 100;
   PLI_ST[136] := 100;
   PLI_ST[137] := 100;
   PLI_ST[138] := 100;
   PLI_ST[139] := 100;
   PLI_ST[140] := 100;
   PLI_ST[141] := 100;
   PLI_ST[142] := 100;
   PLI_ST[143] := 100;
   PLI_ST[144] := 100;
   PLI_ST[145] := 100;
   PLI_ST[146] := 100;
   PLI_ST[147] := 100;
   PLI_ST[148] := 100;
   PLI_ST[149] := 100;
   PLI_ST[150] := 100;
   PLI_SI[1] := 1;
   PLI_SI[2] := 1;
   PLI_SI[3] := 1;
   PLI_SI[4] := 1;
   PLI_SI[5] := 1;
   PLI_SI[6] := 1;
   PLI_SI[7] := 1;
   PLI_SI[8] := 1;
   PLI_SI[9] := 1;
   PLI_SI[10] := 1;
   PLI_SI[11] := 1;
   PLI_SI[12] := 1;
   PLI_SI[13] := 1;
   PLI_SI[14] := 1;
   PLI_SI[15] := 1;
   PLI_SI[16] := 1;
   PLI_SI[17] := 1;
   PLI_SI[18] := 1;
   PLI_SI[19] := 1;
   PLI_SI[20] := 1;
   PLI_SI[21] := 1;
   PLI_SI[22] := 1;
   PLI_SI[23] := 1;
   PLI_SI[24] := 1;
   PLI_SI[25] := 1;
   PLI_SI[26] := 1;
   PLI_SI[27] := 1;
   PLI_SI[28] := 1;
   PLI_SI[29] := 1;
   PLI_SI[30] := 1;
   PLI_SI[31] := 1;
   PLI_SI[32] := 1;
   PLI_SI[33] := 1;
   PLI_SI[34] := 1;
   PLI_SI[35] := 1;
   PLI_SI[36] := 1;
   PLI_SI[37] := 1;
   PLI_SI[38] := 1;
   PLI_SI[39] := 1;
   PLI_SI[40] := 1;
   PLI_SI[41] := 1;
   PLI_SI[42] := 1;
   PLI_SI[43] := 1;
   PLI_SI[44] := 1;
   PLI_SI[45] := 1;
   PLI_SI[46] := 1;
   PLI_SI[47] := 1;
   PLI_SI[48] := 1;
   PLI_SI[49] := 1;
   PLI_SI[50] := 1;
   PLI_SI[51] := 1;
   PLI_SI[52] := 1;
   PLI_SI[53] := 1;
   PLI_SI[54] := 1;
   PLI_SI[55] := 1;
   PLI_SI[56] := 1;
   PLI_SI[57] := 1;
   PLI_SI[58] := 1;
   PLI_SI[59] := 1;
   PLI_SI[60] := 1;
   PLI_SI[61] := 1;
   PLI_SI[62] := 1;
   PLI_SI[63] := 1;
   PLI_SI[64] := 1;
   PLI_SI[65] := 1;
   PLI_SI[66] := 1;
   PLI_SI[67] := 1;
   PLI_SI[68] := 1;
   PLI_SI[69] := 1;
   PLI_SI[70] := 1;
   PLI_SI[71] := 1;
   PLI_SI[72] := 1;
   PLI_SI[73] := 1;
   PLI_SI[74] := 1;
   PLI_SI[75] := 1;
   PLI_SI[76] := 1;
   PLI_SI[77] := 1;
   PLI_SI[78] := 1;
   PLI_SI[79] := 1;
   PLI_SI[80] := 1;
   PLI_SI[81] := 1;
   PLI_SI[82] := 1;
   PLI_SI[83] := 1;
   PLI_SI[84] := 1;
   PLI_SI[85] := 1;
   PLI_SI[86] := 1;
   PLI_SI[87] := 1;
   PLI_SI[88] := 1;
   PLI_SI[89] := 1;
   PLI_SI[90] := 1;
   PLI_SI[91] := 1;
   PLI_SI[92] := 1;
   PLI_SI[93] := 1;
   PLI_SI[94] := 1;
   PLI_SI[95] := 1;
   PLI_SI[96] := 1;
   PLI_SI[97] := 1;
   PLI_SI[98] := 1;
   PLI_SI[99] := 1;
   PLI_SI[100] := 1;
   PLI_SI[101] := 1;
   PLI_SI[102] := 1;
   PLI_SI[103] := 1;
   PLI_SI[104] := 1;
   PLI_SI[105] := 1;
   PLI_SI[106] := 1;
   PLI_SI[107] := 1;
   PLI_SI[108] := 1;
   PLI_SI[109] := 1;
   PLI_SI[110] := 100;
   PLI_SI[111] := 10;
   PLI_SI[112] := 1;
   PLI_SI[113] := 1;
   PLI_SI[114] := 1;
   PLI_SI[115] := 1;
   PLI_SI[116] := 200;
   PLI_SI[117] := 1;
   PLI_SI[118] := 1;
   PLI_SI[119] := 1;
   PLI_SI[120] := 1;
   PLI_SI[121] := 1;
   PLI_SI[122] := 1;
   PLI_SI[123] := 1;
   PLI_SI[124] := 1;
   PLI_SI[125] := 1;
   PLI_SI[126] := 1;
   PLI_SI[127] := 1;
   PLI_SI[128] := 1;
   PLI_SI[129] := 1;
   PLI_SI[130] := 1;
   PLI_SI[131] := 1;
   PLI_SI[132] := 1;
   PLI_SI[133] := 1;
   PLI_SI[134] := 1;
   PLI_SI[135] := 1;
   PLI_SI[136] := 1;
   PLI_SI[137] := 1;
   PLI_SI[138] := 1;
   PLI_SI[139] := 1;
   PLI_SI[140] := 1;
   PLI_SI[141] := 1;
   PLI_SI[142] := 1;
   PLI_SI[143] := 1;
   PLI_SI[144] := 1;
   PLI_SI[145] := 1;
   PLI_SI[146] := 1;
   PLI_SI[147] := 1;
   PLI_SI[148] := 1;
   PLI_SI[149] := 1;
   PLI_SI[150] := 1;
   PLI_OP[1] := 0;
   PLI_OP[2] := 0;
   PLI_OP[3] := 0;
   PLI_OP[4] := 0;
   PLI_OP[5] := 0;
   PLI_OP[6] := 0;
   PLI_OP[7] := 0;
   PLI_OP[8] := 0;
   PLI_OP[9] := 0;
   PLI_OP[10] := 0;
   PLI_OP[11] := 0;
   PLI_OP[12] := 0;
   PLI_OP[13] := 0;
   PLI_OP[14] := 0;
   PLI_OP[15] := 0;
   PLI_OP[16] := 0;
   PLI_OP[17] := 0;
   PLI_OP[18] := 0;
   PLI_OP[19] := 0;
   PLI_OP[20] := 0;
   PLI_OP[21] := 0;
   PLI_OP[22] := 0;
   PLI_OP[23] := 0;
   PLI_OP[24] := 0;
   PLI_OP[25] := 0;
   PLI_OP[26] := 0;
   PLI_OP[27] := 0;
   PLI_OP[28] := 0;
   PLI_OP[29] := 0;
   PLI_OP[30] := 0;
   PLI_OP[31] := 0;
   PLI_OP[32] := 0;
   PLI_OP[33] := 0;
   PLI_OP[34] := 0;
   PLI_OP[35] := 0;
   PLI_OP[36] := 0;
   PLI_OP[37] := 0;
   PLI_OP[38] := 0;
   PLI_OP[39] := 0;
   PLI_OP[40] := 0;
   PLI_OP[41] := 0;
   PLI_OP[42] := 0;
   PLI_OP[43] := 0;
   PLI_OP[44] := 0;
   PLI_OP[45] := 0;
   PLI_OP[46] := 0;
   PLI_OP[47] := 0;
   PLI_OP[48] := 0;
   PLI_OP[49] := 0;
   PLI_OP[50] := 0;
   PLI_OP[51] := 0;
   PLI_OP[52] := 0;
   PLI_OP[53] := 0;
   PLI_OP[54] := 0;
   PLI_OP[55] := 0;
   PLI_OP[56] := 0;
   PLI_OP[57] := 0;
   PLI_OP[58] := 0;
   PLI_OP[59] := 0;
   PLI_OP[60] := 0;
   PLI_OP[61] := 0;
   PLI_OP[62] := 0;
   PLI_OP[63] := 0;
   PLI_OP[64] := 0;
   PLI_OP[65] := 0;
   PLI_OP[66] := 0;
   PLI_OP[67] := 0;
   PLI_OP[68] := 0;
   PLI_OP[69] := 0;
   PLI_OP[70] := 0;
   PLI_OP[71] := 0;
   PLI_OP[72] := 0;
   PLI_OP[73] := 0;
   PLI_OP[74] := 0;
   PLI_OP[75] := 0;
   PLI_OP[76] := 0;
   PLI_OP[77] := 0;
   PLI_OP[78] := 0;
   PLI_OP[79] := 0;
   PLI_OP[80] := 0;
   PLI_OP[81] := 0;
   PLI_OP[82] := 0;
   PLI_OP[83] := 0;
   PLI_OP[84] := 0;
   PLI_OP[85] := 0;
   PLI_OP[86] := 0;
   PLI_OP[87] := 0;
   PLI_OP[88] := 0;
   PLI_OP[89] := 0;
   PLI_OP[90] := 0;
   PLI_OP[91] := 0;
   PLI_OP[92] := -15;
   PLI_OP[93] := 0;
   PLI_OP[94] := 0;
   PLI_OP[95] := 0;
   PLI_OP[96] := 0;
   PLI_OP[97] := 0;
   PLI_OP[98] := 0;
   PLI_OP[99] := 0;
   PLI_OP[100] := 0;
   PLI_OP[101] := 0;
   PLI_OP[102] := 0;
   PLI_OP[103] := 0;
   PLI_OP[104] := 0;
   PLI_OP[105] := 0;
   PLI_OP[106] := 0;
   PLI_OP[107] := 0;
   PLI_OP[108] := 0;
   PLI_OP[109] := 0;
   PLI_OP[110] := 0;
   PLI_OP[111] := 0;
   PLI_OP[112] := 0;
   PLI_OP[113] := 0;
   PLI_OP[114] := 0;
   PLI_OP[115] := 0;
   PLI_OP[116] := 0;
   PLI_OP[117] := 0;
   PLI_OP[118] := 0;
   PLI_OP[119] := 0;
   PLI_OP[120] := 0;
   PLI_OP[121] := 0;
   PLI_OP[122] := 0;
   PLI_OP[123] := 0;
   PLI_OP[124] := 0;
   PLI_OP[125] := 0;
   PLI_OP[126] := 0;
   PLI_OP[127] := 0;
   PLI_OP[128] := 0;
   PLI_OP[129] := 0;
   PLI_OP[130] := 0;
   PLI_OP[131] := 0;
   PLI_OP[132] := 0;
   PLI_OP[133] := 0;
   PLI_OP[134] := 0;
   PLI_OP[135] := 0;
   PLI_OP[136] := 0;
   PLI_OP[137] := 0;
   PLI_OP[138] := 0;
   PLI_OP[139] := 0;
   PLI_OP[140] := 0;
   PLI_OP[141] := 0;
   PLI_OP[142] := 0;
   PLI_OP[143] := 0;
   PLI_OP[144] := 0;
   PLI_OP[145] := 0;
   PLI_OP[146] := 0;
   PLI_OP[147] := 0;
   PLI_OP[148] := 0;
   PLI_OP[149] := 0;
   PLI_OP[150] := 0;
   PLI_WR[1] := 16#0000;
   PLI_WR[2] := 16#0000;
   PLI_WR[3] := 16#0000;
   PLI_WR[4] := 16#0000;
   PLI_WR[5] := 16#0000;
   PLI_WR[6] := 16#0000;
   PLI_WR[7] := 16#0000;
   PLI_WR[8] := 16#0000;
   PLI_WR[9] := 16#0000;
   PLI_WR[10] := 16#0000;
   PLI_WR[11] := 16#0000;
   PLI_WR[12] := 16#0000;
   PLI_WR[13] := 16#0000;
   PLI_WR[14] := 16#0000;
   PLI_WR[15] := 16#0000;
   PLI_WR[16] := 16#0000;
   PLI_WR[17] := 16#0000;
   PLI_WR[18] := 16#0000;
   PLI_WR[19] := 16#0000;
   PLI_WR[20] := 16#0000;
   PLI_WR[21] := 16#0000;
   PLI_WR[22] := 16#0000;
   PLI_WR[23] := 16#0000;
   PLI_WR[24] := 16#0000;
   PLI_WR[25] := 16#0000;
   PLI_WR[26] := 16#0000;
   PLI_WR[27] := 16#0000;
   PLI_WR[28] := 16#0000;
   PLI_WR[29] := 16#0000;
   PLI_WR[30] := 16#0000;
   PLI_WR[31] := 16#0000;
   PLI_WR[32] := 16#0000;
   PLI_WR[33] := 16#0000;
   PLI_WR[34] := 16#0000;
   PLI_WR[35] := 16#0000;
   PLI_WR[36] := 16#0000;
   PLI_WR[37] := 16#0000;
   PLI_WR[38] := 16#0000;
   PLI_WR[39] := 16#0000;
   PLI_WR[40] := 16#0000;
   PLI_WR[41] := 16#0000;
   PLI_WR[42] := 16#0000;
   PLI_WR[43] := 16#0000;
   PLI_WR[44] := 16#0000;
   PLI_WR[45] := 16#0000;
   PLI_WR[46] := 16#0000;
   PLI_WR[47] := 16#0000;
   PLI_WR[48] := 16#0000;
   PLI_WR[49] := 16#0000;
   PLI_WR[50] := 16#0000;
   PLI_WR[51] := 16#0000;
   PLI_WR[52] := 16#0000;
   PLI_WR[53] := 16#0000;
   PLI_WR[54] := 16#0000;
   PLI_WR[55] := 16#0000;
   PLI_WR[56] := 16#0000;
   PLI_WR[57] := 16#0000;
   PLI_WR[58] := 16#0000;
   PLI_WR[59] := 16#0000;
   PLI_WR[60] := 16#0000;
   PLI_WR[61] := 16#0000;
   PLI_WR[62] := 16#0000;
   PLI_WR[63] := 16#0000;
   PLI_WR[64] := 16#0000;
   PLI_WR[65] := 16#0000;
   PLI_WR[66] := 16#0000;
   PLI_WR[67] := 16#0000;
   PLI_WR[68] := 16#0000;
   PLI_WR[69] := 16#0000;
   PLI_WR[70] := 16#0000;
   PLI_WR[71] := 16#0000;
   PLI_WR[72] := 16#0000;
   PLI_WR[73] := 16#0000;
   PLI_WR[74] := 16#0000;
   PLI_WR[75] := 16#0000;
   PLI_WR[76] := 16#0000;
   PLI_WR[77] := 16#0000;
   PLI_WR[78] := 16#0000;
   PLI_WR[79] := 16#0000;
   PLI_WR[80] := 16#0000;
   PLI_WR[81] := 16#0000;
   PLI_WR[82] := 16#0000;
   PLI_WR[83] := 16#0000;
   PLI_WR[84] := 16#0000;
   PLI_WR[85] := 16#0000;
   PLI_WR[86] := 16#0000;
   PLI_WR[87] := 16#0000;
   PLI_WR[88] := 16#0000;
   PLI_WR[89] := 16#0000;
   PLI_WR[90] := 16#0000;
   PLI_WR[91] := 16#0000;
   PLI_WR[92] := 16#0000;
   PLI_WR[93] := 16#0000;
   PLI_WR[94] := 16#0000;
   PLI_WR[95] := 16#0000;
   PLI_WR[96] := 16#0000;
   PLI_WR[97] := 16#0000;
   PLI_WR[98] := 16#0000;
   PLI_WR[99] := 16#0000;
   PLI_WR[100] := 16#0000;
   PLI_WR[101] := 16#0000;
   PLI_WR[102] := 16#0000;
   PLI_WR[103] := 16#0000;
   PLI_WR[104] := 16#0000;
   PLI_WR[105] := 16#0000;
   PLI_WR[106] := 16#0000;
   PLI_WR[107] := 16#0000;
   PLI_WR[108] := 16#0000;
   PLI_WR[109] := 16#0000;
   PLI_WR[110] := 16#0000;
   PLI_WR[111] := 16#0000;
   PLI_WR[112] := 16#0000;
   PLI_WR[113] := 16#0000;
   PLI_WR[114] := 16#0000;
   PLI_WR[115] := 16#0000;
   PLI_WR[116] := 16#0000;
   PLI_WR[117] := 16#0000;
   PLI_WR[118] := 16#0000;
   PLI_WR[119] := 16#0000;
   PLI_WR[120] := 16#0000;
   PLI_WR[121] := 16#0000;
   PLI_WR[122] := 16#0000;
   PLI_WR[123] := 16#0000;
   PLI_WR[124] := 16#0000;
   PLI_WR[125] := 16#0000;
   PLI_WR[126] := 16#0000;
   PLI_WR[127] := 16#0000;
   PLI_WR[128] := 16#0000;
   PLI_WR[129] := 16#0000;
   PLI_WR[130] := 16#0000;
   PLI_WR[131] := 16#0000;
   PLI_WR[132] := 16#0000;
   PLI_WR[133] := 16#0000;
   PLI_WR[134] := 16#0000;
   PLI_WR[135] := 16#0000;
   PLI_WR[136] := 16#0000;
   PLI_WR[137] := 16#0000;
   PLI_WR[138] := 16#0000;
   PLI_WR[139] := 16#0000;
   PLI_WR[140] := 16#0000;
   PLI_WR[141] := 16#0000;
   PLI_WR[142] := 16#0000;
   PLI_WR[143] := 16#0000;
   PLI_WR[144] := 16#0000;
   PLI_WR[145] := 16#0000;
   PLI_WR[146] := 16#0000;
   PLI_WR[147] := 16#0000;
   PLI_WR[148] := 16#0000;
   PLI_WR[149] := 16#0000;
   PLI_WR[150] := 16#0000;
   PLI_OC[1] := 0;
   PLI_OC[2] := 0;
   PLI_OC[3] := 0;
   PLI_OC[4] := 0;
   PLI_OC[5] := 0;
   PLI_OC[6] := 0;
   PLI_OC[7] := 0;
   PLI_OC[8] := 0;
   PLI_OC[9] := 0;
   PLI_OC[10] := 0;
   PLI_OC[11] := 0;
   PLI_OC[12] := 0;
   PLI_OC[13] := 0;
   PLI_OC[14] := 0;
   PLI_OC[15] := 0;
   PLI_OC[16] := 0;
   PLI_OC[17] := 0;
   PLI_OC[18] := 0;
   PLI_OC[19] := 0;
   PLI_OC[20] := 0;
   PLI_OC[21] := 0;
   PLI_OC[22] := 0;
   PLI_OC[23] := 0;
   PLI_OC[24] := 0;
   PLI_OC[25] := 0;
   PLI_OC[26] := 0;
   PLI_OC[27] := 0;
   PLI_OC[28] := 0;
   PLI_OC[29] := 0;
   PLI_OC[30] := 0;
   PLI_OC[31] := 0;
   PLI_OC[32] := 0;
   PLI_OC[33] := 0;
   PLI_OC[34] := 0;
   PLI_OC[35] := 0;
   PLI_OC[36] := 0;
   PLI_OC[37] := 0;
   PLI_OC[38] := 0;
   PLI_OC[39] := 0;
   PLI_OC[40] := 0;
   PLI_OC[41] := 0;
   PLI_OC[42] := 0;
   PLI_OC[43] := 0;
   PLI_OC[44] := 0;
   PLI_OC[45] := 0;
   PLI_OC[46] := 0;
   PLI_OC[47] := 0;
   PLI_OC[48] := 0;
   PLI_OC[49] := 0;
   PLI_OC[50] := 0;
   PLI_OC[51] := 0;
   PLI_OC[52] := 0;
   PLI_OC[53] := 0;
   PLI_OC[54] := 0;
   PLI_OC[55] := 0;
   PLI_OC[56] := 0;
   PLI_OC[57] := 0;
   PLI_OC[58] := 0;
   PLI_OC[59] := 0;
   PLI_OC[60] := 0;
   PLI_OC[61] := 0;
   PLI_OC[62] := 0;
   PLI_OC[63] := 0;
   PLI_OC[64] := 0;
   PLI_OC[65] := 0;
   PLI_OC[66] := 0;
   PLI_OC[67] := 0;
   PLI_OC[68] := 0;
   PLI_OC[69] := 0;
   PLI_OC[70] := 0;
   PLI_OC[71] := 0;
   PLI_OC[72] := 0;
   PLI_OC[73] := 0;
   PLI_OC[74] := 0;
   PLI_OC[75] := 0;
   PLI_OC[76] := 0;
   PLI_OC[77] := 0;
   PLI_OC[78] := 0;
   PLI_OC[79] := 0;
   PLI_OC[80] := 0;
   PLI_OC[81] := 0;
   PLI_OC[82] := 0;
   PLI_OC[83] := 0;
   PLI_OC[84] := 0;
   PLI_OC[85] := 0;
   PLI_OC[86] := 0;
   PLI_OC[87] := 0;
   PLI_OC[88] := 0;
   PLI_OC[89] := 0;
   PLI_OC[90] := 0;
   PLI_OC[91] := 0;
   PLI_OC[92] := 0;
   PLI_OC[93] := 0;
   PLI_OC[94] := 0;
   PLI_OC[95] := 0;
   PLI_OC[96] := 0;
   PLI_OC[97] := 0;
   PLI_OC[98] := 0;
   PLI_OC[99] := 0;
   PLI_OC[100] := 0;
   PLI_OC[101] := 0;
   PLI_OC[102] := 0;
   PLI_OC[103] := 0;
   PLI_OC[104] := 0;
   PLI_OC[105] := 0;
   PLI_OC[106] := 0;
   PLI_OC[107] := 0;
   PLI_OC[108] := 0;
   PLI_OC[109] := 0;
   PLI_OC[110] := 0;
   PLI_OC[111] := 0;
   PLI_OC[112] := 0;
   PLI_OC[113] := 0;
   PLI_OC[114] := 0;
   PLI_OC[115] := 0;
   PLI_OC[116] := 0;
   PLI_OC[117] := 0;
   PLI_OC[118] := 0;
   PLI_OC[119] := 0;
   PLI_OC[120] := 0;
   PLI_OC[121] := 0;
   PLI_OC[122] := 0;
   PLI_OC[123] := 0;
   PLI_OC[124] := 0;
   PLI_OC[125] := 0;
   PLI_OC[126] := 0;
   PLI_OC[127] := 0;
   PLI_OC[128] := 0;
   PLI_OC[129] := 0;
   PLI_OC[130] := 0;
   PLI_OC[131] := 0;
   PLI_OC[132] := 0;
   PLI_OC[133] := 0;
   PLI_OC[134] := 0;
   PLI_OC[135] := 0;
   PLI_OC[136] := 0;
   PLI_OC[137] := 0;
   PLI_OC[138] := 0;
   PLI_OC[139] := 0;
   PLI_OC[140] := 0;
   PLI_OC[141] := 0;
   PLI_OC[142] := 0;
   PLI_OC[143] := 0;
   PLI_OC[144] := 0;
   PLI_OC[145] := 0;
   PLI_OC[146] := 0;
   PLI_OC[147] := 0;
   PLI_OC[148] := 0;
   PLI_OC[149] := 0;
   PLI_OC[150] := 0;
   PLI_CD[1] := 0;
   PLI_CD[2] := 0;
   PLI_CD[3] := 0;
   PLI_CD[4] := 0;
   PLI_CD[5] := 0;
   PLI_CD[6] := 0;
   PLI_CD[7] := 0;
   PLI_CD[8] := 0;
   PLI_CD[9] := 0;
   PLI_CD[10] := 0;
   PLI_CD[11] := 0;
   PLI_CD[12] := 0;
   PLI_CD[13] := 0;
   PLI_CD[14] := 0;
   PLI_CD[15] := 0;
   PLI_CD[16] := 0;
   PLI_CD[17] := 0;
   PLI_CD[18] := 0;
   PLI_CD[19] := 0;
   PLI_CD[20] := 0;
   PLI_CD[21] := 0;
   PLI_CD[22] := 0;
   PLI_CD[23] := 0;
   PLI_CD[24] := 0;
   PLI_CD[25] := 0;
   PLI_CD[26] := 0;
   PLI_CD[27] := 0;
   PLI_CD[28] := 0;
   PLI_CD[29] := 0;
   PLI_CD[30] := 0;
   PLI_CD[31] := 0;
   PLI_CD[32] := 0;
   PLI_CD[33] := 0;
   PLI_CD[34] := 0;
   PLI_CD[35] := 0;
   PLI_CD[36] := 0;
   PLI_CD[37] := 0;
   PLI_CD[38] := 0;
   PLI_CD[39] := 0;
   PLI_CD[40] := 0;
   PLI_CD[41] := 0;
   PLI_CD[42] := 0;
   PLI_CD[43] := 0;
   PLI_CD[44] := 0;
   PLI_CD[45] := 0;
   PLI_CD[46] := 0;
   PLI_CD[47] := 0;
   PLI_CD[48] := 0;
   PLI_CD[49] := 0;
   PLI_CD[50] := 0;
   PLI_CD[51] := 0;
   PLI_CD[52] := 0;
   PLI_CD[53] := 0;
   PLI_CD[54] := 0;
   PLI_CD[55] := 0;
   PLI_CD[56] := 0;
   PLI_CD[57] := 0;
   PLI_CD[58] := 0;
   PLI_CD[59] := 0;
   PLI_CD[60] := 0;
   PLI_CD[61] := 0;
   PLI_CD[62] := 0;
   PLI_CD[63] := 0;
   PLI_CD[64] := 0;
   PLI_CD[65] := 0;
   PLI_CD[66] := 0;
   PLI_CD[67] := 0;
   PLI_CD[68] := 0;
   PLI_CD[69] := 0;
   PLI_CD[70] := 0;
   PLI_CD[71] := 0;
   PLI_CD[72] := 0;
   PLI_CD[73] := 0;
   PLI_CD[74] := 0;
   PLI_CD[75] := 0;
   PLI_CD[76] := 0;
   PLI_CD[77] := 0;
   PLI_CD[78] := 0;
   PLI_CD[79] := 0;
   PLI_CD[80] := 0;
   PLI_CD[81] := 0;
   PLI_CD[82] := 0;
   PLI_CD[83] := 0;
   PLI_CD[84] := 0;
   PLI_CD[85] := 0;
   PLI_CD[86] := 0;
   PLI_CD[87] := 0;
   PLI_CD[88] := 0;
   PLI_CD[89] := 0;
   PLI_CD[90] := 0;
   PLI_CD[91] := 0;
   PLI_CD[92] := 0;
   PLI_CD[93] := 0;
   PLI_CD[94] := 0;
   PLI_CD[95] := 0;
   PLI_CD[96] := 0;
   PLI_CD[97] := 0;
   PLI_CD[98] := 0;
   PLI_CD[99] := 0;
   PLI_CD[100] := 0;
   PLI_CD[101] := 0;
   PLI_CD[102] := 0;
   PLI_CD[103] := 0;
   PLI_CD[104] := 0;
   PLI_CD[105] := 0;
   PLI_CD[106] := 0;
   PLI_CD[107] := 0;
   PLI_CD[108] := 0;
   PLI_CD[109] := 0;
   PLI_CD[110] := 0;
   PLI_CD[111] := 0;
   PLI_CD[112] := 0;
   PLI_CD[113] := 0;
   PLI_CD[114] := 0;
   PLI_CD[115] := 0;
   PLI_CD[116] := 0;
   PLI_CD[117] := 0;
   PLI_CD[118] := 0;
   PLI_CD[119] := 0;
   PLI_CD[120] := 0;
   PLI_CD[121] := 0;
   PLI_CD[122] := 0;
   PLI_CD[123] := 0;
   PLI_CD[124] := 0;
   PLI_CD[125] := 0;
   PLI_CD[126] := 0;
   PLI_CD[127] := 0;
   PLI_CD[128] := 0;
   PLI_CD[129] := 0;
   PLI_CD[130] := 0;
   PLI_CD[131] := 0;
   PLI_CD[132] := 0;
   PLI_CD[133] := 0;
   PLI_CD[134] := 0;
   PLI_CD[135] := 0;
   PLI_CD[136] := 0;
   PLI_CD[137] := 0;
   PLI_CD[138] := 0;
   PLI_CD[139] := 0;
   PLI_CD[140] := 0;
   PLI_CD[141] := 0;
   PLI_CD[142] := 0;
   PLI_CD[143] := 0;
   PLI_CD[144] := 0;
   PLI_CD[145] := 0;
   PLI_CD[146] := 0;
   PLI_CD[147] := 0;
   PLI_CD[148] := 0;
   PLI_CD[149] := 0;
   PLI_CD[150] := 0;
   PLI_IS[1] := 0;
   PLI_IS[2] := 0;
   PLI_IS[3] := 0;
   PLI_IS[4] := 0;
   PLI_IS[5] := 0;
   PLI_IS[6] := 0;
   PLI_IS[7] := 0;
   PLI_IS[8] := 0;
   PLI_IS[9] := 0;
   PLI_IS[10] := 0;
   PLI_IS[11] := 0;
   PLI_IS[12] := 0;
   PLI_IS[13] := 0;
   PLI_IS[14] := 0;
   PLI_IS[15] := 0;
   PLI_IS[16] := 0;
   PLI_IS[17] := 0;
   PLI_IS[18] := 0;
   PLI_IS[19] := 0;
   PLI_IS[20] := 0;
   PLI_IS[21] := 0;
   PLI_IS[22] := 0;
   PLI_IS[23] := 0;
   PLI_IS[24] := 0;
   PLI_IS[25] := 0;
   PLI_IS[26] := 0;
   PLI_IS[27] := 0;
   PLI_IS[28] := 0;
   PLI_IS[29] := 0;
   PLI_IS[30] := 0;
   PLI_IS[31] := 0;
   PLI_IS[32] := 0;
   PLI_IS[33] := 0;
   PLI_IS[34] := 0;
   PLI_IS[35] := 0;
   PLI_IS[36] := 0;
   PLI_IS[37] := 0;
   PLI_IS[38] := 0;
   PLI_IS[39] := 0;
   PLI_IS[40] := 0;
   PLI_IS[41] := 0;
   PLI_IS[42] := 0;
   PLI_IS[43] := 0;
   PLI_IS[44] := 0;
   PLI_IS[45] := 0;
   PLI_IS[46] := 0;
   PLI_IS[47] := 0;
   PLI_IS[48] := 0;
   PLI_IS[49] := 0;
   PLI_IS[50] := 0;
   PLI_IS[51] := 0;
   PLI_IS[52] := 0;
   PLI_IS[53] := 0;
   PLI_IS[54] := 0;
   PLI_IS[55] := 0;
   PLI_IS[56] := 0;
   PLI_IS[57] := 0;
   PLI_IS[58] := 0;
   PLI_IS[59] := 0;
   PLI_IS[60] := 0;
   PLI_IS[61] := 0;
   PLI_IS[62] := 0;
   PLI_IS[63] := 0;
   PLI_IS[64] := 0;
   PLI_IS[65] := 0;
   PLI_IS[66] := 0;
   PLI_IS[67] := 0;
   PLI_IS[68] := 0;
   PLI_IS[69] := 0;
   PLI_IS[70] := 0;
   PLI_IS[71] := 0;
   PLI_IS[72] := 0;
   PLI_IS[73] := 0;
   PLI_IS[74] := 0;
   PLI_IS[75] := 0;
   PLI_IS[76] := 0;
   PLI_IS[77] := 0;
   PLI_IS[78] := 0;
   PLI_IS[79] := 0;
   PLI_IS[80] := 0;
   PLI_IS[81] := 0;
   PLI_IS[82] := 0;
   PLI_IS[83] := 0;
   PLI_IS[84] := 0;
   PLI_IS[85] := 0;
   PLI_IS[86] := 0;
   PLI_IS[87] := 0;
   PLI_IS[88] := 0;
   PLI_IS[89] := 0;
   PLI_IS[90] := 0;
   PLI_IS[91] := 0;
   PLI_IS[92] := 0;
   PLI_IS[93] := 0;
   PLI_IS[94] := 0;
   PLI_IS[95] := 0;
   PLI_IS[96] := 0;
   PLI_IS[97] := 0;
   PLI_IS[98] := 0;
   PLI_IS[99] := 0;
   PLI_IS[100] := 0;
   PLI_IS[101] := 0;
   PLI_IS[102] := 0;
   PLI_IS[103] := 0;
   PLI_IS[104] := 0;
   PLI_IS[105] := 0;
   PLI_IS[106] := 0;
   PLI_IS[107] := 0;
   PLI_IS[108] := 0;
   PLI_IS[109] := 0;
   PLI_IS[110] := 0;
   PLI_IS[111] := 0;
   PLI_IS[112] := 0;
   PLI_IS[113] := 0;
   PLI_IS[114] := 0;
   PLI_IS[115] := 0;
   PLI_IS[116] := 0;
   PLI_IS[117] := 0;
   PLI_IS[118] := 0;
   PLI_IS[119] := 0;
   PLI_IS[120] := 0;
   PLI_IS[121] := 0;
   PLI_IS[122] := 0;
   PLI_IS[123] := 0;
   PLI_IS[124] := 0;
   PLI_IS[125] := 0;
   PLI_IS[126] := 0;
   PLI_IS[127] := 0;
   PLI_IS[128] := 0;
   PLI_IS[129] := 0;
   PLI_IS[130] := 0;
   PLI_IS[131] := 0;
   PLI_IS[132] := 0;
   PLI_IS[133] := 0;
   PLI_IS[134] := 0;
   PLI_IS[135] := 0;
   PLI_IS[136] := 0;
   PLI_IS[137] := 0;
   PLI_IS[138] := 0;
   PLI_IS[139] := 0;
   PLI_IS[140] := 0;
   PLI_IS[141] := 0;
   PLI_IS[142] := 0;
   PLI_IS[143] := 0;
   PLI_IS[144] := 0;
   PLI_IS[145] := 0;
   PLI_IS[146] := 0;
   PLI_IS[147] := 0;
   PLI_IS[148] := 0;
   PLI_IS[149] := 0;
   PLI_IS[150] := 0;
   PLI_UN[1] := 1;
   PLI_UN[2] := 1;
   PLI_UN[3] := 1;
   PLI_UN[4] := 1;
   PLI_UN[5] := 1;
   PLI_UN[6] := 1;
   PLI_UN[7] := 1;
   PLI_UN[8] := 1;
   PLI_UN[9] := 1;
   PLI_UN[10] := 1;
   PLI_UN[11] := 1;
   PLI_UN[12] := 1;
   PLI_UN[13] := 1;
   PLI_UN[14] := 1;
   PLI_UN[15] := 1;
   PLI_UN[16] := 1;
   PLI_UN[17] := 1;
   PLI_UN[18] := 1;
   PLI_UN[19] := 1;
   PLI_UN[20] := 1;
   PLI_UN[21] := 1;
   PLI_UN[22] := 1;
   PLI_UN[23] := 1;
   PLI_UN[24] := 1;
   PLI_UN[25] := 1;
   PLI_UN[26] := 1;
   PLI_UN[27] := 1;
   PLI_UN[28] := 1;
   PLI_UN[29] := 1;
   PLI_UN[30] := 1;
   PLI_UN[31] := 1;
   PLI_UN[32] := 1;
   PLI_UN[33] := 1;
   PLI_UN[34] := 1;
   PLI_UN[35] := 1;
   PLI_UN[36] := 1;
   PLI_UN[37] := 1;
   PLI_UN[38] := 1;
   PLI_UN[39] := 1;
   PLI_UN[40] := 1;
   PLI_UN[41] := 1;
   PLI_UN[42] := 1;
   PLI_UN[43] := 1;
   PLI_UN[44] := 1;
   PLI_UN[45] := 1;
   PLI_UN[46] := 1;
   PLI_UN[47] := 1;
   PLI_UN[48] := 1;
   PLI_UN[49] := 1;
   PLI_UN[50] := 1;
   PLI_UN[51] := 1;
   PLI_UN[52] := 1;
   PLI_UN[53] := 1;
   PLI_UN[54] := 1;
   PLI_UN[55] := 1;
   PLI_UN[56] := 1;
   PLI_UN[57] := 1;
   PLI_UN[58] := 1;
   PLI_UN[59] := 1;
   PLI_UN[60] := 1;
   PLI_UN[61] := 1;
   PLI_UN[62] := 1;
   PLI_UN[63] := 1;
   PLI_UN[64] := 1;
   PLI_UN[65] := 1;
   PLI_UN[66] := 1;
   PLI_UN[67] := 1;
   PLI_UN[68] := 1;
   PLI_UN[69] := 1;
   PLI_UN[70] := 1;
   PLI_UN[71] := 1;
   PLI_UN[72] := 1;
   PLI_UN[73] := 1;
   PLI_UN[74] := 1;
   PLI_UN[75] := 1;
   PLI_UN[76] := 1;
   PLI_UN[77] := 1;
   PLI_UN[78] := 1;
   PLI_UN[79] := 1;
   PLI_UN[80] := 1;
   PLI_UN[81] := 1;
   PLI_UN[82] := 1;
   PLI_UN[83] := 1;
   PLI_UN[84] := 1;
   PLI_UN[85] := 1;
   PLI_UN[86] := 1;
   PLI_UN[87] := 1;
   PLI_UN[88] := 1;
   PLI_UN[89] := 1;
   PLI_UN[90] := 1;
   PLI_UN[91] := 1;
   PLI_UN[92] := 1;
   PLI_UN[93] := 1;
   PLI_UN[94] := 1;
   PLI_UN[95] := 1;
   PLI_UN[96] := 1;
   PLI_UN[97] := 1;
   PLI_UN[98] := 1;
   PLI_UN[99] := 1;
   PLI_UN[100] := 1;
   PLI_UN[101] := 1;
   PLI_UN[102] := 1;
   PLI_UN[103] := 1;
   PLI_UN[104] := 1;
   PLI_UN[105] := 1;
   PLI_UN[106] := 1;
   PLI_UN[107] := 1;
   PLI_UN[108] := 1;
   PLI_UN[109] := 1;
   PLI_UN[110] := 1;
   PLI_UN[111] := 1;
   PLI_UN[112] := 1;
   PLI_UN[113] := 1;
   PLI_UN[114] := 1;
   PLI_UN[115] := 1;
   PLI_UN[116] := 1;
   PLI_UN[117] := 1;
   PLI_UN[118] := 1;
   PLI_UN[119] := 1;
   PLI_UN[120] := 1;
   PLI_UN[121] := 1;
   PLI_UN[122] := 9;
   PLI_UN[123] := 9;
   PLI_UN[124] := 0;
   PLI_UN[125] := 0;
   PLI_UN[126] := 0;
   PLI_UN[127] := 0;
   PLI_UN[128] := 0;
   PLI_UN[129] := 0;
   PLI_UN[130] := 0;
   PLI_UN[131] := 0;
   PLI_UN[132] := 0;
   PLI_UN[133] := 0;
   PLI_UN[134] := 0;
   PLI_UN[135] := 0;
   PLI_UN[136] := 0;
   PLI_UN[137] := 0;
   PLI_UN[138] := 0;
   PLI_UN[139] := 0;
   PLI_UN[140] := 0;
   PLI_UN[141] := 0;
   PLI_UN[142] := 0;
   PLI_UN[143] := 0;
   PLI_UN[144] := 0;
   PLI_UN[145] := 0;
   PLI_UN[146] := 0;
   PLI_UN[147] := 0;
   PLI_UN[148] := 0;
   PLI_UN[149] := 0;
   PLI_UN[150] := 0;
   PLI_F[1] := 0;
   PLI_F[2] := 0;
   PLI_F[3] := 0;
   PLI_F[4] := 0;
   PLI_F[5] := 0;
   PLI_F[6] := 0;
   PLI_F[7] := 0;
   PLI_F[8] := 0;
   PLI_F[9] := 0;
   PLI_F[10] := 0;
   PLI_F[11] := 0;
   PLI_F[12] := 0;
   PLI_F[13] := 0;
   PLI_F[14] := 0;
   PLI_F[15] := 0;
   PLI_F[16] := 0;
   PLI_F[17] := 0;
   PLI_F[18] := 0;
   PLI_F[19] := 0;
   PLI_F[20] := 0;
   PLI_F[21] := 0;
   PLI_F[22] := 0;
   PLI_F[23] := 0;
   PLI_F[24] := 0;
   PLI_F[25] := 0;
   PLI_F[26] := 0;
   PLI_F[27] := 0;
   PLI_F[28] := 0;
   PLI_F[29] := 0;
   PLI_F[30] := 0;
   PLI_F[31] := 0;
   PLI_F[32] := 0;
   PLI_F[33] := 0;
   PLI_F[34] := 0;
   PLI_F[35] := 0;
   PLI_F[36] := 0;
   PLI_F[37] := 0;
   PLI_F[38] := 0;
   PLI_F[39] := 0;
   PLI_F[40] := 0;
   PLI_F[41] := 0;
   PLI_F[42] := 0;
   PLI_F[43] := 0;
   PLI_F[44] := 0;
   PLI_F[45] := 0;
   PLI_F[46] := 0;
   PLI_F[47] := 0;
   PLI_F[48] := 0;
   PLI_F[49] := 0;
   PLI_F[50] := 0;
   PLI_F[51] := 0;
   PLI_F[52] := 0;
   PLI_F[53] := 0;
   PLI_F[54] := 0;
   PLI_F[55] := 0;
   PLI_F[56] := 0;
   PLI_F[57] := 0;
   PLI_F[58] := 0;
   PLI_F[59] := 0;
   PLI_F[60] := 0;
   PLI_F[61] := 0;
   PLI_F[62] := 0;
   PLI_F[63] := 0;
   PLI_F[64] := 0;
   PLI_F[65] := 0;
   PLI_F[66] := 0;
   PLI_F[67] := 0;
   PLI_F[68] := 0;
   PLI_F[69] := 0;
   PLI_F[70] := 0;
   PLI_F[71] := 0;
   PLI_F[72] := 0;
   PLI_F[73] := 0;
   PLI_F[74] := 0;
   PLI_F[75] := 0;
   PLI_F[76] := 0;
   PLI_F[77] := 0;
   PLI_F[78] := 0;
   PLI_F[79] := 0;
   PLI_F[80] := 0;
   PLI_F[81] := 0;
   PLI_F[82] := 0;
   PLI_F[83] := 0;
   PLI_F[84] := 0;
   PLI_F[85] := 0;
   PLI_F[86] := 0;
   PLI_F[87] := 0;
   PLI_F[88] := 0;
   PLI_F[89] := 0;
   PLI_F[90] := 0;
   PLI_F[91] := 0;
   PLI_F[92] := 0;
   PLI_F[93] := 0;
   PLI_F[94] := 0;
   PLI_F[95] := 0;
   PLI_F[96] := 0;
   PLI_F[97] := 0;
   PLI_F[98] := 0;
   PLI_F[99] := 0;
   PLI_F[100] := 0;
   PLI_F[101] := 0;
   PLI_F[102] := 0;
   PLI_F[103] := 0;
   PLI_F[104] := 0;
   PLI_F[105] := 0;
   PLI_F[106] := 0;
   PLI_F[107] := 0;
   PLI_F[108] := 0;
   PLI_F[109] := 0;
   PLI_F[110] := 0;
   PLI_F[111] := 0;
   PLI_F[112] := 0;
   PLI_F[113] := 0;
   PLI_F[114] := 0;
   PLI_F[115] := 0;
   PLI_F[116] := 0;
   PLI_F[117] := 0;
   PLI_F[118] := 0;
   PLI_F[119] := 0;
   PLI_F[120] := 0;
   PLI_F[121] := 0;
   PLI_F[122] := 0;
   PLI_F[123] := 0;
   PLI_F[124] := 0;
   PLI_F[125] := 0;
   PLI_F[126] := 0;
   PLI_F[127] := 0;
   PLI_F[128] := 0;
   PLI_F[129] := 0;
   PLI_F[130] := 0;
   PLI_F[131] := 0;
   PLI_F[132] := 0;
   PLI_F[133] := 0;
   PLI_F[134] := 0;
   PLI_F[135] := 0;
   PLI_F[136] := 0;
   PLI_F[137] := 0;
   PLI_F[138] := 0;
   PLI_F[139] := 0;
   PLI_F[140] := 0;
   PLI_F[141] := 0;
   PLI_F[142] := 0;
   PLI_F[143] := 0;
   PLI_F[144] := 0;
   PLI_F[145] := 0;
   PLI_F[146] := 0;
   PLI_F[147] := 0;
   PLI_F[148] := 0;
   PLI_F[149] := 0;
   PLI_F[150] := 0;
   PLI_RQ[1] := 0;
   PLI_RQ[2] := 0;
   PLI_RQ[3] := 0;
   PLI_RQ[4] := 0;
   PLI_RQ[5] := 0;
   PLI_RQ[6] := 0;
   PLI_RQ[7] := 0;
   PLI_RQ[8] := 0;
   PLI_RQ[9] := 0;
   PLI_RQ[10] := 0;
   PLI_RQ[11] := 0;
   PLI_RQ[12] := 0;
   PLI_RQ[13] := 0;
   PLI_RQ[14] := 0;
   PLI_RQ[15] := 0;
   PLI_RQ[16] := 0;
   PLI_RQ[17] := 0;
   PLI_RQ[18] := 0;
   PLI_RQ[19] := 0;
   PLI_RQ[20] := 0;
   PLI_RQ[21] := 0;
   PLI_RQ[22] := 0;
   PLI_RQ[23] := 0;
   PLI_RQ[24] := 0;
   PLI_RQ[25] := 0;
   PLI_RQ[26] := 0;
   PLI_RQ[27] := 0;
   PLI_RQ[28] := 0;
   PLI_RQ[29] := 0;
   PLI_RQ[30] := 0;
   PLI_RQ[31] := 0;
   PLI_RQ[32] := 0;
   PLI_RQ[33] := 0;
   PLI_RQ[34] := 0;
   PLI_RQ[35] := 0;
   PLI_RQ[36] := 0;
   PLI_RQ[37] := 0;
   PLI_RQ[38] := 0;
   PLI_RQ[39] := 0;
   PLI_RQ[40] := 0;
   PLI_RQ[41] := 0;
   PLI_RQ[42] := 0;
   PLI_RQ[43] := 0;
   PLI_RQ[44] := 0;
   PLI_RQ[45] := 0;
   PLI_RQ[46] := 0;
   PLI_RQ[47] := 0;
   PLI_RQ[48] := 0;
   PLI_RQ[49] := 0;
   PLI_RQ[50] := 0;
   PLI_RQ[51] := 0;
   PLI_RQ[52] := 0;
   PLI_RQ[53] := 0;
   PLI_RQ[54] := 0;
   PLI_RQ[55] := 0;
   PLI_RQ[56] := 0;
   PLI_RQ[57] := 0;
   PLI_RQ[58] := 0;
   PLI_RQ[59] := 0;
   PLI_RQ[60] := 0;
   PLI_RQ[61] := 0;
   PLI_RQ[62] := 0;
   PLI_RQ[63] := 0;
   PLI_RQ[64] := 0;
   PLI_RQ[65] := 0;
   PLI_RQ[66] := 0;
   PLI_RQ[67] := 0;
   PLI_RQ[68] := 0;
   PLI_RQ[69] := 0;
   PLI_RQ[70] := 0;
   PLI_RQ[71] := 0;
   PLI_RQ[72] := 0;
   PLI_RQ[73] := 0;
   PLI_RQ[74] := 0;
   PLI_RQ[75] := 0;
   PLI_RQ[76] := 0;
   PLI_RQ[77] := 0;
   PLI_RQ[78] := 0;
   PLI_RQ[79] := 0;
   PLI_RQ[80] := 0;
   PLI_RQ[81] := 0;
   PLI_RQ[82] := 0;
   PLI_RQ[83] := 0;
   PLI_RQ[84] := 0;
   PLI_RQ[85] := 0;
   PLI_RQ[86] := 0;
   PLI_RQ[87] := 0;
   PLI_RQ[88] := 0;
   PLI_RQ[89] := 0;
   PLI_RQ[90] := 0;
   PLI_RQ[91] := 0;
   PLI_RQ[92] := 0;
   PLI_RQ[93] := 0;
   PLI_RQ[94] := 0;
   PLI_RQ[95] := 0;
   PLI_RQ[96] := 0;
   PLI_RQ[97] := 0;
   PLI_RQ[98] := 0;
   PLI_RQ[99] := 0;
   PLI_RQ[100] := 0;
   PLI_RQ[101] := 0;
   PLI_RQ[102] := 0;
   PLI_RQ[103] := 0;
   PLI_RQ[104] := 0;
   PLI_RQ[105] := 0;
   PLI_RQ[106] := 0;
   PLI_RQ[107] := 0;
   PLI_RQ[108] := 0;
   PLI_RQ[109] := 0;
   PLI_RQ[110] := 0;
   PLI_RQ[111] := 0;
   PLI_RQ[112] := 0;
   PLI_RQ[113] := 0;
   PLI_RQ[114] := 0;
   PLI_RQ[115] := 0;
   PLI_RQ[116] := 0;
   PLI_RQ[117] := 0;
   PLI_RQ[118] := 0;
   PLI_RQ[119] := 0;
   PLI_RQ[120] := 0;
   PLI_RQ[121] := 0;
   PLI_RQ[122] := 0;
   PLI_RQ[123] := 0;
   PLI_RQ[124] := 0;
   PLI_RQ[125] := 0;
   PLI_RQ[126] := 0;
   PLI_RQ[127] := 0;
   PLI_RQ[128] := 0;
   PLI_RQ[129] := 0;
   PLI_RQ[130] := 0;
   PLI_RQ[131] := 0;
   PLI_RQ[132] := 0;
   PLI_RQ[133] := 0;
   PLI_RQ[134] := 0;
   PLI_RQ[135] := 0;
   PLI_RQ[136] := 0;
   PLI_RQ[137] := 0;
   PLI_RQ[138] := 0;
   PLI_RQ[139] := 0;
   PLI_RQ[140] := 0;
   PLI_RQ[141] := 0;
   PLI_RQ[142] := 0;
   PLI_RQ[143] := 0;
   PLI_RQ[144] := 0;
   PLI_RQ[145] := 0;
   PLI_RQ[146] := 0;
   PLI_RQ[147] := 0;
   PLI_RQ[148] := 0;
   PLI_RQ[149] := 0;
   PLI_RQ[150] := 0;
   PLI_SB[1] := 100;
   PLI_SB[2] := 5;
   PLI_SB[3] := 10;
   PLI_SB[4] := 140;
   PLI_SB[5] := 100;
   PLI_SB[6] := 30;
   PLI_SB[7] := 320;
   PLI_SB[8] := 10;
   PLI_SB[9] := 100;
   PLI_SB[10] := 100;
   PLI_SB[11] := 10;
   PLI_SB[12] := 100;
   PLI_SB[13] := 10;
   PLI_SB[14] := 10;
   PLI_SB[15] := 10;
   PLI_SB[16] := 100;
   PLI_SB[17] := 10;
   PLI_SB[18] := 10;
   PLI_SB[19] := 10;
   PLI_SB[20] := 100;
   PLI_SB[21] := 100;
   PLI_SB[22] := 30;
   PLI_SB[23] := 10;
   PLI_SB[24] := 10;
   PLI_SB[25] := 100;
   PLI_SB[26] := 10;
   PLI_SB[27] := 10;
   PLI_SB[28] := 10;
   PLI_SB[29] := 100;
   PLI_SB[30] := 100;
   PLI_SB[31] := 150;
   PLI_SB[32] := 10;
   PLI_SB[33] := 5;
   PLI_SB[34] := 105;
   PLI_SB[35] := 5;
   PLI_SB[36] := 10;
   PLI_SB[37] := 10;
   PLI_SB[38] := 80;
   PLI_SB[39] := 100;
   PLI_SB[40] := 100;
   PLI_SB[41] := 100;
   PLI_SB[42] := 10;
   PLI_SB[43] := 10;
   PLI_SB[44] := 30;
   PLI_SB[45] := 100;
   PLI_SB[46] := 100;
   PLI_SB[47] := 60;
   PLI_SB[48] := 20;
   PLI_SB[49] := 10;
   PLI_SB[50] := 100;
   PLI_SB[51] := 2;
   PLI_SB[52] := 220;
   PLI_SB[53] := 100;
   PLI_SB[54] := 140;
   PLI_SB[55] := 10;
   PLI_SB[56] := 0;
   PLI_SB[57] := 100;
   PLI_SB[58] := 100;
   PLI_SB[59] := 100;
   PLI_SB[60] := 100;
   PLI_SB[61] := 20;
   PLI_SB[62] := 30;
   PLI_SB[63] := 10;
   PLI_SB[64] := 100;
   PLI_SB[65] := 5;
   PLI_SB[66] := 20;
   PLI_SB[67] := 10;
   PLI_SB[68] := 5;
   PLI_SB[69] := 30;
   PLI_SB[70] := 100;
   PLI_SB[71] := 100;
   PLI_SB[72] := 30;
   PLI_SB[73] := 15;
   PLI_SB[74] := 5;
   PLI_SB[75] := 100;
   PLI_SB[76] := 20;
   PLI_SB[77] := 10;
   PLI_SB[78] := 20;
   PLI_SB[79] := 100;
   PLI_SB[80] := 5;
   PLI_SB[81] := 100;
   PLI_SB[82] := 100;
   PLI_SB[83] := 10;
   PLI_SB[84] := 10;
   PLI_SB[85] := 100;
   PLI_SB[86] := 100;
   PLI_SB[87] := 100;
   PLI_SB[88] := 100;
   PLI_SB[89] := 10;
   PLI_SB[90] := 400;
   PLI_SB[91] := 10;
   PLI_SB[92] := 10;
   PLI_SB[93] := 10;
   PLI_SB[94] := 100;
   PLI_SB[95] := 13;
   PLI_SB[96] := 60;
   PLI_SB[97] := 0;
   PLI_SB[98] := 1;
   PLI_SB[99] := 0;
   PLI_SB[100] := 9;
   PLI_SB[101] := 10;
   PLI_SB[102] := 10;
   PLI_SB[103] := 10;
   PLI_SB[104] := 0;
   PLI_SB[105] := 400;
   PLI_SB[106] := 0;
   PLI_SB[107] := 0;
   PLI_SB[108] := 0;
   PLI_SB[109] := 0;
   PLI_SB[110] := 100;
   PLI_SB[111] := 5;
   PLI_SB[112] := 0;
   PLI_SB[113] := 0;
   PLI_SB[114] := 0;
   PLI_SB[115] := 0;
   PLI_SB[116] := 0;
   PLI_SB[117] := 0;
   PLI_SB[118] := 0;
   PLI_SB[119] := 0;
   PLI_SB[120] := 100;
   PLI_SB[121] := 20;
   PLI_SB[122] := 1;
   PLI_SB[123] := 0;
   PLI_SB[124] := 0;
   PLI_SB[125] := 0;
   PLI_SB[126] := 0;
   PLI_SB[127] := 0;
   PLI_SB[128] := 0;
   PLI_SB[129] := 0;
   PLI_SB[130] := 0;
   PLI_SB[131] := 0;
   PLI_SB[132] := 0;
   PLI_SB[133] := 0;
   PLI_SB[134] := 0;
   PLI_SB[135] := 0;
   PLI_SB[136] := 0;
   PLI_SB[137] := 0;
   PLI_SB[138] := 0;
   PLI_SB[139] := 0;
   PLI_SB[140] := 0;
   PLI_SB[141] := 0;
   PLI_SB[142] := 0;
   PLI_SB[143] := 0;
   PLI_SB[144] := 0;
   PLI_SB[145] := 0;
   PLI_SB[146] := 0;
   PLI_SB[147] := 0;
   PLI_SB[148] := 0;
   PLI_SB[149] := 0;
   PLI_SB[150] := 0;
   PLI_BRQ[1] := 0;
   PLI_BRQ[2] := 0;
   PLI_BRQ[3] := 0;
   PLI_BRQ[4] := 0;
   PLI_BRQ[5] := 0;
   PLI_BRQ[6] := 0;
   PLI_BRQ[7] := 0;
   PLI_BRQ[8] := 0;
   PLI_BRQ[9] := 0;
   PLI_BRQ[10] := 0;
   PLI_BRQ[11] := 0;
   PLI_BRQ[12] := 0;
   PLI_BRQ[13] := 0;
   PLI_BRQ[14] := 0;
   PLI_BRQ[15] := 0;
   PLI_BRQ[16] := 0;
   PLI_BRQ[17] := 0;
   PLI_BRQ[18] := 0;
   PLI_BRQ[19] := 0;
   PLI_BRQ[20] := 0;
   PLI_BRQ[21] := 0;
   PLI_BRQ[22] := 0;
   PLI_BRQ[23] := 0;
   PLI_BRQ[24] := 0;
   PLI_BRQ[25] := 0;
   PLI_BRQ[26] := 0;
   PLI_BRQ[27] := 0;
   PLI_BRQ[28] := 0;
   PLI_BRQ[29] := 0;
   PLI_BRQ[30] := 0;
   PLI_BRQ[31] := 0;
   PLI_BRQ[32] := 0;
   PLI_BRQ[33] := 0;
   PLI_BRQ[34] := 0;
   PLI_BRQ[35] := 0;
   PLI_BRQ[36] := 0;
   PLI_BRQ[37] := 0;
   PLI_BRQ[38] := 0;
   PLI_BRQ[39] := 0;
   PLI_BRQ[40] := 0;
   PLI_BRQ[41] := 0;
   PLI_BRQ[42] := 0;
   PLI_BRQ[43] := 0;
   PLI_BRQ[44] := 0;
   PLI_BRQ[45] := 0;
   PLI_BRQ[46] := 0;
   PLI_BRQ[47] := 0;
   PLI_BRQ[48] := 0;
   PLI_BRQ[49] := 0;
   PLI_BRQ[50] := 0;
   PLI_BRQ[51] := 0;
   PLI_BRQ[52] := 0;
   PLI_BRQ[53] := 0;
   PLI_BRQ[54] := 0;
   PLI_BRQ[55] := 0;
   PLI_BRQ[56] := 0;
   PLI_BRQ[57] := 0;
   PLI_BRQ[58] := 0;
   PLI_BRQ[59] := 0;
   PLI_BRQ[60] := 0;
   PLI_BRQ[61] := 0;
   PLI_BRQ[62] := 0;
   PLI_BRQ[63] := 0;
   PLI_BRQ[64] := 0;
   PLI_BRQ[65] := 0;
   PLI_BRQ[66] := 0;
   PLI_BRQ[67] := 0;
   PLI_BRQ[68] := 0;
   PLI_BRQ[69] := 0;
   PLI_BRQ[70] := 0;
   PLI_BRQ[71] := 0;
   PLI_BRQ[72] := 0;
   PLI_BRQ[73] := 0;
   PLI_BRQ[74] := 0;
   PLI_BRQ[75] := 0;
   PLI_BRQ[76] := 0;
   PLI_BRQ[77] := 0;
   PLI_BRQ[78] := 0;
   PLI_BRQ[79] := 0;
   PLI_BRQ[80] := 0;
   PLI_BRQ[81] := 0;
   PLI_BRQ[82] := 0;
   PLI_BRQ[83] := 0;
   PLI_BRQ[84] := 0;
   PLI_BRQ[85] := 0;
   PLI_BRQ[86] := 0;
   PLI_BRQ[87] := 0;
   PLI_BRQ[88] := 0;
   PLI_BRQ[89] := 0;
   PLI_BRQ[90] := 0;
   PLI_BRQ[91] := 0;
   PLI_BRQ[92] := 0;
   PLI_BRQ[93] := 0;
   PLI_BRQ[94] := 0;
   PLI_BRQ[95] := 0;
   PLI_BRQ[96] := 0;
   PLI_BRQ[97] := 0;
   PLI_BRQ[98] := 0;
   PLI_BRQ[99] := 0;
   PLI_BRQ[100] := 0;
   PLI_BRQ[101] := 0;
   PLI_BRQ[102] := 0;
   PLI_BRQ[103] := 0;
   PLI_BRQ[104] := 0;
   PLI_BRQ[105] := 0;
   PLI_BRQ[106] := 0;
   PLI_BRQ[107] := 0;
   PLI_BRQ[108] := 0;
   PLI_BRQ[109] := 0;
   PLI_BRQ[110] := 0;
   PLI_BRQ[111] := 0;
   PLI_BRQ[112] := 0;
   PLI_BRQ[113] := 0;
   PLI_BRQ[114] := 0;
   PLI_BRQ[115] := 0;
   PLI_BRQ[116] := 0;
   PLI_BRQ[117] := 0;
   PLI_BRQ[118] := 0;
   PLI_BRQ[119] := 0;
   PLI_BRQ[120] := 0;
   PLI_BRQ[121] := 0;
   PLI_BRQ[122] := 0;
   PLI_BRQ[123] := 0;
   PLI_BRQ[124] := 0;
   PLI_BRQ[125] := 0;
   PLI_BRQ[126] := 0;
   PLI_BRQ[127] := 0;
   PLI_BRQ[128] := 0;
   PLI_BRQ[129] := 0;
   PLI_BRQ[130] := 0;
   PLI_BRQ[131] := 0;
   PLI_BRQ[132] := 0;
   PLI_BRQ[133] := 0;
   PLI_BRQ[134] := 0;
   PLI_BRQ[135] := 0;
   PLI_BRQ[136] := 0;
   PLI_BRQ[137] := 0;
   PLI_BRQ[138] := 0;
   PLI_BRQ[139] := 0;
   PLI_BRQ[140] := 0;
   PLI_BRQ[141] := 0;
   PLI_BRQ[142] := 0;
   PLI_BRQ[143] := 0;
   PLI_BRQ[144] := 0;
   PLI_BRQ[145] := 0;
   PLI_BRQ[146] := 0;
   PLI_BRQ[147] := 0;
   PLI_BRQ[148] := 0;
   PLI_BRQ[149] := 0;
   PLI_BRQ[150] := 0;
   PLI_HI[1] := 30;
   PLI_HI[2] := 10;
   PLI_HI[3] := 30;
   PLI_HI[4] := 30;
   PLI_HI[5] := 10;
   PLI_HI[6] := 10;
   PLI_HI[7] := 10;
   PLI_HI[8] := 10;
   PLI_HI[9] := 10;
   PLI_HI[10] := 10;
   PLI_HI[11] := 10;
   PLI_HI[12] := 30;
   PLI_HI[13] := 10;
   PLI_HI[14] := 10;
   PLI_HI[15] := 10;
   PLI_HI[16] := 10;
   PLI_HI[17] := 10;
   PLI_HI[18] := 10;
   PLI_HI[19] := 10;
   PLI_HI[20] := 30;
   PLI_HI[21] := 10;
   PLI_HI[22] := 10;
   PLI_HI[23] := 30;
   PLI_HI[24] := 30;
   PLI_HI[25] := 10;
   PLI_HI[26] := 30;
   PLI_HI[27] := 10;
   PLI_HI[28] := 10;
   PLI_HI[29] := 10;
   PLI_HI[30] := 10;
   PLI_HI[31] := 30;
   PLI_HI[32] := 10;
   PLI_HI[33] := 10;
   PLI_HI[34] := 10;
   PLI_HI[35] := 10;
   PLI_HI[36] := 30;
   PLI_HI[37] := 30;
   PLI_HI[38] := 10;
   PLI_HI[39] := 10;
   PLI_HI[40] := 10;
   PLI_HI[41] := 10;
   PLI_HI[42] := 30;
   PLI_HI[43] := 10;
   PLI_HI[44] := 10;
   PLI_HI[45] := 30;
   PLI_HI[46] := 10;
   PLI_HI[47] := 10;
   PLI_HI[48] := 10;
   PLI_HI[49] := 30;
   PLI_HI[50] := 10;
   PLI_HI[51] := 10;
   PLI_HI[52] := 10;
   PLI_HI[53] := 30;
   PLI_HI[54] := 30;
   PLI_HI[55] := 30;
   PLI_HI[56] := 0;
   PLI_HI[57] := 30;
   PLI_HI[58] := 10;
   PLI_HI[59] := 10;
   PLI_HI[60] := 10;
   PLI_HI[61] := 10;
   PLI_HI[62] := 10;
   PLI_HI[63] := 10;
   PLI_HI[64] := 10;
   PLI_HI[65] := 10;
   PLI_HI[66] := 10;
   PLI_HI[67] := 10;
   PLI_HI[68] := 10;
   PLI_HI[69] := 10;
   PLI_HI[70] := 30;
   PLI_HI[71] := 30;
   PLI_HI[72] := 10;
   PLI_HI[73] := 10;
   PLI_HI[74] := 10;
   PLI_HI[75] := 10;
   PLI_HI[76] := 10;
   PLI_HI[77] := 10;
   PLI_HI[78] := 30;
   PLI_HI[79] := 30;
   PLI_HI[80] := 10;
   PLI_HI[81] := 10;
   PLI_HI[82] := 10;
   PLI_HI[83] := 30;
   PLI_HI[84] := 10;
   PLI_HI[85] := 10;
   PLI_HI[86] := 30;
   PLI_HI[87] := 10;
   PLI_HI[88] := 10;
   PLI_HI[89] := 10;
   PLI_HI[90] := 10;
   PLI_HI[91] := 10;
   PLI_HI[92] := 10;
   PLI_HI[93] := 30;
   PLI_HI[94] := 10;
   PLI_HI[95] := 10;
   PLI_HI[96] := 10;
   PLI_HI[97] := 0;
   PLI_HI[98] := 10;
   PLI_HI[99] := 0;
   PLI_HI[100] := 30;
   PLI_HI[101] := 10;
   PLI_HI[102] := 30;
   PLI_HI[103] := 10;
   PLI_HI[104] := 0;
   PLI_HI[105] := 30;
   PLI_HI[106] := 0;
   PLI_HI[107] := 0;
   PLI_HI[108] := 0;
   PLI_HI[109] := 0;
   PLI_HI[110] := 10;
   PLI_HI[111] := 10;
   PLI_HI[112] := 0;
   PLI_HI[113] := 0;
   PLI_HI[114] := 0;
   PLI_HI[115] := 0;
   PLI_HI[116] := 0;
   PLI_HI[117] := 0;
   PLI_HI[118] := 0;
   PLI_HI[119] := 0;
   PLI_HI[120] := 30;
   PLI_HI[121] := 10;
   PLI_HI[122] := 10;
   PLI_HI[123] := 0;
   PLI_HI[124] := 0;
   PLI_HI[125] := 0;
   PLI_HI[126] := 0;
   PLI_HI[127] := 0;
   PLI_HI[128] := 0;
   PLI_HI[129] := 0;
   PLI_HI[130] := 0;
   PLI_HI[131] := 0;
   PLI_HI[132] := 0;
   PLI_HI[133] := 0;
   PLI_HI[134] := 0;
   PLI_HI[135] := 0;
   PLI_HI[136] := 0;
   PLI_HI[137] := 0;
   PLI_HI[138] := 0;
   PLI_HI[139] := 0;
   PLI_HI[140] := 0;
   PLI_HI[141] := 0;
   PLI_HI[142] := 0;
   PLI_HI[143] := 0;
   PLI_HI[144] := 0;
   PLI_HI[145] := 0;
   PLI_HI[146] := 0;
   PLI_HI[147] := 0;
   PLI_HI[148] := 0;
   PLI_HI[149] := 0;
   PLI_HI[150] := 0;
   PLI_MS[1] := 1;
   PLI_MS[2] := 1;
   PLI_MS[3] := 1;
   PLI_MS[4] := 1;
   PLI_MS[5] := 1;
   PLI_MS[6] := 1;
   PLI_MS[7] := 1;
   PLI_MS[8] := 1;
   PLI_MS[9] := 1;
   PLI_MS[10] := 1;
   PLI_MS[11] := 1;
   PLI_MS[12] := 1;
   PLI_MS[13] := 1;
   PLI_MS[14] := 1;
   PLI_MS[15] := 1;
   PLI_MS[16] := 1;
   PLI_MS[17] := 1;
   PLI_MS[18] := 1;
   PLI_MS[19] := 1;
   PLI_MS[20] := 1;
   PLI_MS[21] := 1;
   PLI_MS[22] := 1;
   PLI_MS[23] := 1;
   PLI_MS[24] := 1;
   PLI_MS[25] := 1;
   PLI_MS[26] := 1;
   PLI_MS[27] := 1;
   PLI_MS[28] := 1;
   PLI_MS[29] := 1;
   PLI_MS[30] := 1;
   PLI_MS[31] := 1;
   PLI_MS[32] := 1;
   PLI_MS[33] := 1;
   PLI_MS[34] := 1;
   PLI_MS[35] := 1;
   PLI_MS[36] := 1;
   PLI_MS[37] := 1;
   PLI_MS[38] := 1;
   PLI_MS[39] := 1;
   PLI_MS[40] := 1;
   PLI_MS[41] := 1;
   PLI_MS[42] := 1;
   PLI_MS[43] := 1;
   PLI_MS[44] := 3;
   PLI_MS[45] := 1;
   PLI_MS[46] := 1;
   PLI_MS[47] := 1;
   PLI_MS[48] := 1;
   PLI_MS[49] := 1;
   PLI_MS[50] := 1;
   PLI_MS[51] := 1;
   PLI_MS[52] := 1;
   PLI_MS[53] := 1;
   PLI_MS[54] := 1;
   PLI_MS[55] := 1;
   PLI_MS[56] := 1;
   PLI_MS[57] := 1;
   PLI_MS[58] := 1;
   PLI_MS[59] := 1;
   PLI_MS[60] := 1;
   PLI_MS[61] := 1;
   PLI_MS[62] := 1;
   PLI_MS[63] := 1;
   PLI_MS[64] := 1;
   PLI_MS[65] := 1;
   PLI_MS[66] := 2;
   PLI_MS[67] := 2;
   PLI_MS[68] := 1;
   PLI_MS[69] := 1;
   PLI_MS[70] := 1;
   PLI_MS[71] := 1;
   PLI_MS[72] := 1;
   PLI_MS[73] := 2;
   PLI_MS[74] := 1;
   PLI_MS[75] := 1;
   PLI_MS[76] := 2;
   PLI_MS[77] := 1;
   PLI_MS[78] := 1;
   PLI_MS[79] := 1;
   PLI_MS[80] := 1;
   PLI_MS[81] := 1;
   PLI_MS[82] := 1;
   PLI_MS[83] := 1;
   PLI_MS[84] := 1;
   PLI_MS[85] := 1;
   PLI_MS[86] := 1;
   PLI_MS[87] := 1;
   PLI_MS[88] := 1;
   PLI_MS[89] := 1;
   PLI_MS[90] := 1;
   PLI_MS[91] := 1;
   PLI_MS[92] := 1;
   PLI_MS[93] := 1;
   PLI_MS[94] := 1;
   PLI_MS[95] := 1;
   PLI_MS[96] := 1;
   PLI_MS[97] := 1;
   PLI_MS[98] := 1;
   PLI_MS[99] := 1;
   PLI_MS[100] := 1;
   PLI_MS[101] := 1;
   PLI_MS[102] := 1;
   PLI_MS[103] := 1;
   PLI_MS[104] := 1;
   PLI_MS[105] := 1;
   PLI_MS[106] := 1;
   PLI_MS[107] := 1;
   PLI_MS[108] := 1;
   PLI_MS[109] := 1;
   PLI_MS[110] := 2;
   PLI_MS[111] := 2;
   PLI_MS[112] := 1;
   PLI_MS[113] := 1;
   PLI_MS[114] := 1;
   PLI_MS[115] := 1;
   PLI_MS[116] := 2;
   PLI_MS[117] := 1;
   PLI_MS[118] := 1;
   PLI_MS[119] := 1;
   PLI_MS[120] := 1;
   PLI_MS[121] := 1;
   PLI_MS[122] := 1;
   PLI_MS[123] := 1;
   PLI_MS[124] := 1;
   PLI_MS[125] := 1;
   PLI_MS[126] := 1;
   PLI_MS[127] := 1;
   PLI_MS[128] := 1;
   PLI_MS[129] := 1;
   PLI_MS[130] := 1;
   PLI_MS[131] := 1;
   PLI_MS[132] := 1;
   PLI_MS[133] := 1;
   PLI_MS[134] := 1;
   PLI_MS[135] := 1;
   PLI_MS[136] := 1;
   PLI_MS[137] := 1;
   PLI_MS[138] := 1;
   PLI_MS[139] := 1;
   PLI_MS[140] := 1;
   PLI_MS[141] := 1;
   PLI_MS[142] := 1;
   PLI_MS[143] := 1;
   PLI_MS[144] := 1;
   PLI_MS[145] := 1;
   PLI_MS[146] := 1;
   PLI_MS[147] := 1;
   PLI_MS[148] := 1;
   PLI_MS[149] := 1;
   PLI_MS[150] := 1;
   PLI_MD[1] := 0;
   PLI_MD[2] := 0;
   PLI_MD[3] := 0;
   PLI_MD[4] := 0;
   PLI_MD[5] := 0;
   PLI_MD[6] := 0;
   PLI_MD[7] := 0;
   PLI_MD[8] := 0;
   PLI_MD[9] := 0;
   PLI_MD[10] := 0;
   PLI_MD[11] := 0;
   PLI_MD[12] := 0;
   PLI_MD[13] := 0;
   PLI_MD[14] := 0;
   PLI_MD[15] := 0;
   PLI_MD[16] := 0;
   PLI_MD[17] := 0;
   PLI_MD[18] := 0;
   PLI_MD[19] := 0;
   PLI_MD[20] := 0;
   PLI_MD[21] := 0;
   PLI_MD[22] := 0;
   PLI_MD[23] := 0;
   PLI_MD[24] := 0;
   PLI_MD[25] := 0;
   PLI_MD[26] := 0;
   PLI_MD[27] := 0;
   PLI_MD[28] := 0;
   PLI_MD[29] := 0;
   PLI_MD[30] := 0;
   PLI_MD[31] := 0;
   PLI_MD[32] := 0;
   PLI_MD[33] := 0;
   PLI_MD[34] := 0;
   PLI_MD[35] := 0;
   PLI_MD[36] := 0;
   PLI_MD[37] := 0;
   PLI_MD[38] := 0;
   PLI_MD[39] := 0;
   PLI_MD[40] := 0;
   PLI_MD[41] := 0;
   PLI_MD[42] := 0;
   PLI_MD[43] := 0;
   PLI_MD[44] := 0;
   PLI_MD[45] := 0;
   PLI_MD[46] := 0;
   PLI_MD[47] := 0;
   PLI_MD[48] := 0;
   PLI_MD[49] := 0;
   PLI_MD[50] := 0;
   PLI_MD[51] := 0;
   PLI_MD[52] := 0;
   PLI_MD[53] := 0;
   PLI_MD[54] := 0;
   PLI_MD[55] := 0;
   PLI_MD[56] := 0;
   PLI_MD[57] := 0;
   PLI_MD[58] := 0;
   PLI_MD[59] := 0;
   PLI_MD[60] := 0;
   PLI_MD[61] := 0;
   PLI_MD[62] := 0;
   PLI_MD[63] := 0;
   PLI_MD[64] := 0;
   PLI_MD[65] := 0;
   PLI_MD[66] := 0;
   PLI_MD[67] := 0;
   PLI_MD[68] := 0;
   PLI_MD[69] := 0;
   PLI_MD[70] := 0;
   PLI_MD[71] := 0;
   PLI_MD[72] := 0;
   PLI_MD[73] := 0;
   PLI_MD[74] := 0;
   PLI_MD[75] := 0;
   PLI_MD[76] := 0;
   PLI_MD[77] := 0;
   PLI_MD[78] := 0;
   PLI_MD[79] := 0;
   PLI_MD[80] := 0;
   PLI_MD[81] := 0;
   PLI_MD[82] := 0;
   PLI_MD[83] := 0;
   PLI_MD[84] := 0;
   PLI_MD[85] := 0;
   PLI_MD[86] := 0;
   PLI_MD[87] := 0;
   PLI_MD[88] := 0;
   PLI_MD[89] := 0;
   PLI_MD[90] := 0;
   PLI_MD[91] := 0;
   PLI_MD[92] := 0;
   PLI_MD[93] := 0;
   PLI_MD[94] := 0;
   PLI_MD[95] := 0;
   PLI_MD[96] := 0;
   PLI_MD[97] := 0;
   PLI_MD[98] := 0;
   PLI_MD[99] := 0;
   PLI_MD[100] := 0;
   PLI_MD[101] := 0;
   PLI_MD[102] := 0;
   PLI_MD[103] := 0;
   PLI_MD[104] := 0;
   PLI_MD[105] := 0;
   PLI_MD[106] := 0;
   PLI_MD[107] := 0;
   PLI_MD[108] := 0;
   PLI_MD[109] := 0;
   PLI_MD[110] := 0;
   PLI_MD[111] := 0;
   PLI_MD[112] := 0;
   PLI_MD[113] := 0;
   PLI_MD[114] := 0;
   PLI_MD[115] := 0;
   PLI_MD[116] := 0;
   PLI_MD[117] := 0;
   PLI_MD[118] := 0;
   PLI_MD[119] := 0;
   PLI_MD[120] := 0;
   PLI_MD[121] := 0;
   PLI_MD[122] := 0;
   PLI_MD[123] := 0;
   PLI_MD[124] := 0;
   PLI_MD[125] := 0;
   PLI_MD[126] := 0;
   PLI_MD[127] := 0;
   PLI_MD[128] := 0;
   PLI_MD[129] := 0;
   PLI_MD[130] := 0;
   PLI_MD[131] := 0;
   PLI_MD[132] := 0;
   PLI_MD[133] := 0;
   PLI_MD[134] := 0;
   PLI_MD[135] := 0;
   PLI_MD[136] := 0;
   PLI_MD[137] := 0;
   PLI_MD[138] := 0;
   PLI_MD[139] := 0;
   PLI_MD[140] := 0;
   PLI_MD[141] := 0;
   PLI_MD[142] := 0;
   PLI_MD[143] := 0;
   PLI_MD[144] := 0;
   PLI_MD[145] := 0;
   PLI_MD[146] := 0;
   PLI_MD[147] := 0;
   PLI_MD[148] := 0;
   PLI_MD[149] := 0;
   PLI_MD[150] := 0;
   PLI_RC[1] := FALSE;
   PLI_RC[2] := FALSE;
   PLI_RC[3] := FALSE;
   PLI_RC[4] := FALSE;
   PLI_RC[5] := FALSE;
   PLI_RC[6] := FALSE;
   PLI_RC[7] := FALSE;
   PLI_RC[8] := FALSE;
   PLI_RC[9] := FALSE;
   PLI_RC[10] := FALSE;
   PLI_RC[11] := FALSE;
   PLI_RC[12] := FALSE;
   PLI_RC[13] := FALSE;
   PLI_RC[14] := FALSE;
   PLI_RC[15] := FALSE;
   PLI_RC[16] := FALSE;
   PLI_RC[17] := FALSE;
   PLI_RC[18] := FALSE;
   PLI_RC[19] := FALSE;
   PLI_RC[20] := FALSE;
   PLI_RC[21] := FALSE;
   PLI_RC[22] := FALSE;
   PLI_RC[23] := FALSE;
   PLI_RC[24] := FALSE;
   PLI_RC[25] := FALSE;
   PLI_RC[26] := FALSE;
   PLI_RC[27] := FALSE;
   PLI_RC[28] := FALSE;
   PLI_RC[29] := FALSE;
   PLI_RC[30] := FALSE;
   PLI_RC[31] := FALSE;
   PLI_RC[32] := FALSE;
   PLI_RC[33] := FALSE;
   PLI_RC[34] := FALSE;
   PLI_RC[35] := FALSE;
   PLI_RC[36] := FALSE;
   PLI_RC[37] := FALSE;
   PLI_RC[38] := FALSE;
   PLI_RC[39] := FALSE;
   PLI_RC[40] := FALSE;
   PLI_RC[41] := FALSE;
   PLI_RC[42] := FALSE;
   PLI_RC[43] := FALSE;
   PLI_RC[44] := FALSE;
   PLI_RC[45] := FALSE;
   PLI_RC[46] := FALSE;
   PLI_RC[47] := FALSE;
   PLI_RC[48] := FALSE;
   PLI_RC[49] := FALSE;
   PLI_RC[50] := FALSE;
   PLI_RC[51] := FALSE;
   PLI_RC[52] := FALSE;
   PLI_RC[53] := FALSE;
   PLI_RC[54] := FALSE;
   PLI_RC[55] := FALSE;
   PLI_RC[56] := FALSE;
   PLI_RC[57] := FALSE;
   PLI_RC[58] := FALSE;
   PLI_RC[59] := FALSE;
   PLI_RC[60] := FALSE;
   PLI_RC[61] := FALSE;
   PLI_RC[62] := FALSE;
   PLI_RC[63] := FALSE;
   PLI_RC[64] := FALSE;
   PLI_RC[65] := FALSE;
   PLI_RC[66] := FALSE;
   PLI_RC[67] := FALSE;
   PLI_RC[68] := FALSE;
   PLI_RC[69] := FALSE;
   PLI_RC[70] := FALSE;
   PLI_RC[71] := FALSE;
   PLI_RC[72] := FALSE;
   PLI_RC[73] := FALSE;
   PLI_RC[74] := FALSE;
   PLI_RC[75] := FALSE;
   PLI_RC[76] := FALSE;
   PLI_RC[77] := FALSE;
   PLI_RC[78] := FALSE;
   PLI_RC[79] := FALSE;
   PLI_RC[80] := FALSE;
   PLI_RC[81] := FALSE;
   PLI_RC[82] := FALSE;
   PLI_RC[83] := FALSE;
   PLI_RC[84] := FALSE;
   PLI_RC[85] := FALSE;
   PLI_RC[86] := FALSE;
   PLI_RC[87] := FALSE;
   PLI_RC[88] := FALSE;
   PLI_RC[89] := FALSE;
   PLI_RC[90] := FALSE;
   PLI_RC[91] := FALSE;
   PLI_RC[92] := FALSE;
   PLI_RC[93] := FALSE;
   PLI_RC[94] := FALSE;
   PLI_RC[95] := FALSE;
   PLI_RC[96] := FALSE;
   PLI_RC[97] := FALSE;
   PLI_RC[98] := FALSE;
   PLI_RC[99] := FALSE;
   PLI_RC[100] := FALSE;
   PLI_RC[101] := FALSE;
   PLI_RC[102] := FALSE;
   PLI_RC[103] := FALSE;
   PLI_RC[104] := FALSE;
   PLI_RC[105] := FALSE;
   PLI_RC[106] := FALSE;
   PLI_RC[107] := FALSE;
   PLI_RC[108] := FALSE;
   PLI_RC[109] := FALSE;
   PLI_RC[110] := FALSE;
   PLI_RC[111] := FALSE;
   PLI_RC[112] := FALSE;
   PLI_RC[113] := FALSE;
   PLI_RC[114] := FALSE;
   PLI_RC[115] := FALSE;
   PLI_RC[116] := FALSE;
   PLI_RC[117] := FALSE;
   PLI_RC[118] := FALSE;
   PLI_RC[119] := FALSE;
   PLI_RC[120] := FALSE;
   PLI_RC[121] := FALSE;
   PLI_RC[122] := FALSE;
   PLI_RC[123] := FALSE;
   PLI_RC[124] := FALSE;
   PLI_RC[125] := FALSE;
   PLI_RC[126] := FALSE;
   PLI_RC[127] := FALSE;
   PLI_RC[128] := FALSE;
   PLI_RC[129] := FALSE;
   PLI_RC[130] := FALSE;
   PLI_RC[131] := FALSE;
   PLI_RC[132] := FALSE;
   PLI_RC[133] := FALSE;
   PLI_RC[134] := FALSE;
   PLI_RC[135] := FALSE;
   PLI_RC[136] := FALSE;
   PLI_RC[137] := FALSE;
   PLI_RC[138] := FALSE;
   PLI_RC[139] := FALSE;
   PLI_RC[140] := FALSE;
   PLI_RC[141] := FALSE;
   PLI_RC[142] := FALSE;
   PLI_RC[143] := FALSE;
   PLI_RC[144] := FALSE;
   PLI_RC[145] := FALSE;
   PLI_RC[146] := FALSE;
   PLI_RC[147] := FALSE;
   PLI_RC[148] := FALSE;
   PLI_RC[149] := FALSE;
   PLI_RC[150] := FALSE;
   PLI_TC[1] := FALSE;
   PLI_TC[2] := FALSE;
   PLI_TC[3] := FALSE;
   PLI_TC[4] := FALSE;
   PLI_TC[5] := FALSE;
   PLI_TC[6] := FALSE;
   PLI_TC[7] := FALSE;
   PLI_TC[8] := FALSE;
   PLI_TC[9] := FALSE;
   PLI_TC[10] := FALSE;
   PLI_TC[11] := FALSE;
   PLI_TC[12] := FALSE;
   PLI_TC[13] := FALSE;
   PLI_TC[14] := FALSE;
   PLI_TC[15] := FALSE;
   PLI_TC[16] := FALSE;
   PLI_TC[17] := FALSE;
   PLI_TC[18] := FALSE;
   PLI_TC[19] := FALSE;
   PLI_TC[20] := FALSE;
   PLI_TC[21] := FALSE;
   PLI_TC[22] := FALSE;
   PLI_TC[23] := FALSE;
   PLI_TC[24] := FALSE;
   PLI_TC[25] := FALSE;
   PLI_TC[26] := FALSE;
   PLI_TC[27] := FALSE;
   PLI_TC[28] := FALSE;
   PLI_TC[29] := FALSE;
   PLI_TC[30] := FALSE;
   PLI_TC[31] := FALSE;
   PLI_TC[32] := FALSE;
   PLI_TC[33] := FALSE;
   PLI_TC[34] := FALSE;
   PLI_TC[35] := FALSE;
   PLI_TC[36] := FALSE;
   PLI_TC[37] := FALSE;
   PLI_TC[38] := FALSE;
   PLI_TC[39] := FALSE;
   PLI_TC[40] := FALSE;
   PLI_TC[41] := FALSE;
   PLI_TC[42] := FALSE;
   PLI_TC[43] := FALSE;
   PLI_TC[44] := FALSE;
   PLI_TC[45] := FALSE;
   PLI_TC[46] := FALSE;
   PLI_TC[47] := FALSE;
   PLI_TC[48] := FALSE;
   PLI_TC[49] := FALSE;
   PLI_TC[50] := FALSE;
   PLI_TC[51] := FALSE;
   PLI_TC[52] := FALSE;
   PLI_TC[53] := FALSE;
   PLI_TC[54] := FALSE;
   PLI_TC[55] := FALSE;
   PLI_TC[56] := FALSE;
   PLI_TC[57] := FALSE;
   PLI_TC[58] := FALSE;
   PLI_TC[59] := FALSE;
   PLI_TC[60] := FALSE;
   PLI_TC[61] := FALSE;
   PLI_TC[62] := FALSE;
   PLI_TC[63] := FALSE;
   PLI_TC[64] := FALSE;
   PLI_TC[65] := FALSE;
   PLI_TC[66] := FALSE;
   PLI_TC[67] := FALSE;
   PLI_TC[68] := FALSE;
   PLI_TC[69] := FALSE;
   PLI_TC[70] := FALSE;
   PLI_TC[71] := FALSE;
   PLI_TC[72] := FALSE;
   PLI_TC[73] := FALSE;
   PLI_TC[74] := FALSE;
   PLI_TC[75] := FALSE;
   PLI_TC[76] := FALSE;
   PLI_TC[77] := FALSE;
   PLI_TC[78] := FALSE;
   PLI_TC[79] := FALSE;
   PLI_TC[80] := FALSE;
   PLI_TC[81] := FALSE;
   PLI_TC[82] := FALSE;
   PLI_TC[83] := FALSE;
   PLI_TC[84] := FALSE;
   PLI_TC[85] := FALSE;
   PLI_TC[86] := FALSE;
   PLI_TC[87] := FALSE;
   PLI_TC[88] := FALSE;
   PLI_TC[89] := FALSE;
   PLI_TC[90] := FALSE;
   PLI_TC[91] := FALSE;
   PLI_TC[92] := FALSE;
   PLI_TC[93] := FALSE;
   PLI_TC[94] := FALSE;
   PLI_TC[95] := FALSE;
   PLI_TC[96] := FALSE;
   PLI_TC[97] := FALSE;
   PLI_TC[98] := FALSE;
   PLI_TC[99] := FALSE;
   PLI_TC[100] := FALSE;
   PLI_TC[101] := FALSE;
   PLI_TC[102] := FALSE;
   PLI_TC[103] := FALSE;
   PLI_TC[104] := FALSE;
   PLI_TC[105] := FALSE;
   PLI_TC[106] := FALSE;
   PLI_TC[107] := FALSE;
   PLI_TC[108] := FALSE;
   PLI_TC[109] := FALSE;
   PLI_TC[110] := FALSE;
   PLI_TC[111] := FALSE;
   PLI_TC[112] := FALSE;
   PLI_TC[113] := FALSE;
   PLI_TC[114] := FALSE;
   PLI_TC[115] := FALSE;
   PLI_TC[116] := FALSE;
   PLI_TC[117] := FALSE;
   PLI_TC[118] := FALSE;
   PLI_TC[119] := FALSE;
   PLI_TC[120] := FALSE;
   PLI_TC[121] := FALSE;
   PLI_TC[122] := FALSE;
   PLI_TC[123] := FALSE;
   PLI_TC[124] := FALSE;
   PLI_TC[125] := FALSE;
   PLI_TC[126] := FALSE;
   PLI_TC[127] := FALSE;
   PLI_TC[128] := FALSE;
   PLI_TC[129] := FALSE;
   PLI_TC[130] := FALSE;
   PLI_TC[131] := FALSE;
   PLI_TC[132] := FALSE;
   PLI_TC[133] := FALSE;
   PLI_TC[134] := FALSE;
   PLI_TC[135] := FALSE;
   PLI_TC[136] := FALSE;
   PLI_TC[137] := FALSE;
   PLI_TC[138] := FALSE;
   PLI_TC[139] := FALSE;
   PLI_TC[140] := FALSE;
   PLI_TC[141] := FALSE;
   PLI_TC[142] := FALSE;
   PLI_TC[143] := FALSE;
   PLI_TC[144] := FALSE;
   PLI_TC[145] := FALSE;
   PLI_TC[146] := FALSE;
   PLI_TC[147] := FALSE;
   PLI_TC[148] := FALSE;
   PLI_TC[149] := FALSE;
   PLI_TC[150] := FALSE;
   PLI_AC[1] := FALSE;
   PLI_AC[2] := FALSE;
   PLI_AC[3] := FALSE;
   PLI_AC[4] := FALSE;
   PLI_AC[5] := FALSE;
   PLI_AC[6] := FALSE;
   PLI_AC[7] := FALSE;
   PLI_AC[8] := FALSE;
   PLI_AC[9] := FALSE;
   PLI_AC[10] := FALSE;
   PLI_AC[11] := FALSE;
   PLI_AC[12] := FALSE;
   PLI_AC[13] := FALSE;
   PLI_AC[14] := FALSE;
   PLI_AC[15] := FALSE;
   PLI_AC[16] := FALSE;
   PLI_AC[17] := FALSE;
   PLI_AC[18] := FALSE;
   PLI_AC[19] := FALSE;
   PLI_AC[20] := FALSE;
   PLI_AC[21] := FALSE;
   PLI_AC[22] := FALSE;
   PLI_AC[23] := FALSE;
   PLI_AC[24] := FALSE;
   PLI_AC[25] := FALSE;
   PLI_AC[26] := FALSE;
   PLI_AC[27] := FALSE;
   PLI_AC[28] := FALSE;
   PLI_AC[29] := FALSE;
   PLI_AC[30] := FALSE;
   PLI_AC[31] := FALSE;
   PLI_AC[32] := FALSE;
   PLI_AC[33] := FALSE;
   PLI_AC[34] := FALSE;
   PLI_AC[35] := FALSE;
   PLI_AC[36] := FALSE;
   PLI_AC[37] := FALSE;
   PLI_AC[38] := FALSE;
   PLI_AC[39] := FALSE;
   PLI_AC[40] := FALSE;
   PLI_AC[41] := FALSE;
   PLI_AC[42] := FALSE;
   PLI_AC[43] := FALSE;
   PLI_AC[44] := FALSE;
   PLI_AC[45] := FALSE;
   PLI_AC[46] := FALSE;
   PLI_AC[47] := FALSE;
   PLI_AC[48] := FALSE;
   PLI_AC[49] := FALSE;
   PLI_AC[50] := FALSE;
   PLI_AC[51] := FALSE;
   PLI_AC[52] := FALSE;
   PLI_AC[53] := FALSE;
   PLI_AC[54] := FALSE;
   PLI_AC[55] := FALSE;
   PLI_AC[56] := FALSE;
   PLI_AC[57] := FALSE;
   PLI_AC[58] := FALSE;
   PLI_AC[59] := FALSE;
   PLI_AC[60] := FALSE;
   PLI_AC[61] := FALSE;
   PLI_AC[62] := FALSE;
   PLI_AC[63] := FALSE;
   PLI_AC[64] := FALSE;
   PLI_AC[65] := FALSE;
   PLI_AC[66] := FALSE;
   PLI_AC[67] := FALSE;
   PLI_AC[68] := FALSE;
   PLI_AC[69] := FALSE;
   PLI_AC[70] := FALSE;
   PLI_AC[71] := FALSE;
   PLI_AC[72] := FALSE;
   PLI_AC[73] := FALSE;
   PLI_AC[74] := FALSE;
   PLI_AC[75] := FALSE;
   PLI_AC[76] := FALSE;
   PLI_AC[77] := FALSE;
   PLI_AC[78] := FALSE;
   PLI_AC[79] := FALSE;
   PLI_AC[80] := FALSE;
   PLI_AC[81] := FALSE;
   PLI_AC[82] := FALSE;
   PLI_AC[83] := FALSE;
   PLI_AC[84] := FALSE;
   PLI_AC[85] := FALSE;
   PLI_AC[86] := FALSE;
   PLI_AC[87] := FALSE;
   PLI_AC[88] := FALSE;
   PLI_AC[89] := FALSE;
   PLI_AC[90] := FALSE;
   PLI_AC[91] := FALSE;
   PLI_AC[92] := FALSE;
   PLI_AC[93] := FALSE;
   PLI_AC[94] := FALSE;
   PLI_AC[95] := FALSE;
   PLI_AC[96] := FALSE;
   PLI_AC[97] := FALSE;
   PLI_AC[98] := FALSE;
   PLI_AC[99] := FALSE;
   PLI_AC[100] := FALSE;
   PLI_AC[101] := FALSE;
   PLI_AC[102] := FALSE;
   PLI_AC[103] := FALSE;
   PLI_AC[104] := FALSE;
   PLI_AC[105] := FALSE;
   PLI_AC[106] := FALSE;
   PLI_AC[107] := FALSE;
   PLI_AC[108] := FALSE;
   PLI_AC[109] := FALSE;
   PLI_AC[110] := FALSE;
   PLI_AC[111] := FALSE;
   PLI_AC[112] := FALSE;
   PLI_AC[113] := FALSE;
   PLI_AC[114] := FALSE;
   PLI_AC[115] := FALSE;
   PLI_AC[116] := FALSE;
   PLI_AC[117] := FALSE;
   PLI_AC[118] := FALSE;
   PLI_AC[119] := FALSE;
   PLI_AC[120] := FALSE;
   PLI_AC[121] := FALSE;
   PLI_AC[122] := FALSE;
   PLI_AC[123] := FALSE;
   PLI_AC[124] := FALSE;
   PLI_AC[125] := FALSE;
   PLI_AC[126] := FALSE;
   PLI_AC[127] := FALSE;
   PLI_AC[128] := FALSE;
   PLI_AC[129] := FALSE;
   PLI_AC[130] := FALSE;
   PLI_AC[131] := FALSE;
   PLI_AC[132] := FALSE;
   PLI_AC[133] := FALSE;
   PLI_AC[134] := FALSE;
   PLI_AC[135] := FALSE;
   PLI_AC[136] := FALSE;
   PLI_AC[137] := FALSE;
   PLI_AC[138] := FALSE;
   PLI_AC[139] := FALSE;
   PLI_AC[140] := FALSE;
   PLI_AC[141] := FALSE;
   PLI_AC[142] := FALSE;
   PLI_AC[143] := FALSE;
   PLI_AC[144] := FALSE;
   PLI_AC[145] := FALSE;
   PLI_AC[146] := FALSE;
   PLI_AC[147] := FALSE;
   PLI_AC[148] := FALSE;
   PLI_AC[149] := FALSE;
   PLI_AC[150] := FALSE;
   PLI_HC[1] := FALSE;
   PLI_HC[2] := FALSE;
   PLI_HC[3] := FALSE;
   PLI_HC[4] := FALSE;
   PLI_HC[5] := FALSE;
   PLI_HC[6] := FALSE;
   PLI_HC[7] := FALSE;
   PLI_HC[8] := FALSE;
   PLI_HC[9] := FALSE;
   PLI_HC[10] := FALSE;
   PLI_HC[11] := FALSE;
   PLI_HC[12] := FALSE;
   PLI_HC[13] := FALSE;
   PLI_HC[14] := FALSE;
   PLI_HC[15] := FALSE;
   PLI_HC[16] := FALSE;
   PLI_HC[17] := FALSE;
   PLI_HC[18] := FALSE;
   PLI_HC[19] := FALSE;
   PLI_HC[20] := FALSE;
   PLI_HC[21] := FALSE;
   PLI_HC[22] := FALSE;
   PLI_HC[23] := FALSE;
   PLI_HC[24] := FALSE;
   PLI_HC[25] := FALSE;
   PLI_HC[26] := FALSE;
   PLI_HC[27] := FALSE;
   PLI_HC[28] := FALSE;
   PLI_HC[29] := FALSE;
   PLI_HC[30] := FALSE;
   PLI_HC[31] := FALSE;
   PLI_HC[32] := FALSE;
   PLI_HC[33] := FALSE;
   PLI_HC[34] := FALSE;
   PLI_HC[35] := FALSE;
   PLI_HC[36] := FALSE;
   PLI_HC[37] := FALSE;
   PLI_HC[38] := FALSE;
   PLI_HC[39] := FALSE;
   PLI_HC[40] := FALSE;
   PLI_HC[41] := FALSE;
   PLI_HC[42] := FALSE;
   PLI_HC[43] := FALSE;
   PLI_HC[44] := FALSE;
   PLI_HC[45] := FALSE;
   PLI_HC[46] := FALSE;
   PLI_HC[47] := FALSE;
   PLI_HC[48] := FALSE;
   PLI_HC[49] := FALSE;
   PLI_HC[50] := FALSE;
   PLI_HC[51] := FALSE;
   PLI_HC[52] := FALSE;
   PLI_HC[53] := FALSE;
   PLI_HC[54] := FALSE;
   PLI_HC[55] := FALSE;
   PLI_HC[56] := FALSE;
   PLI_HC[57] := FALSE;
   PLI_HC[58] := FALSE;
   PLI_HC[59] := FALSE;
   PLI_HC[60] := FALSE;
   PLI_HC[61] := FALSE;
   PLI_HC[62] := FALSE;
   PLI_HC[63] := FALSE;
   PLI_HC[64] := FALSE;
   PLI_HC[65] := FALSE;
   PLI_HC[66] := FALSE;
   PLI_HC[67] := FALSE;
   PLI_HC[68] := FALSE;
   PLI_HC[69] := FALSE;
   PLI_HC[70] := FALSE;
   PLI_HC[71] := FALSE;
   PLI_HC[72] := FALSE;
   PLI_HC[73] := FALSE;
   PLI_HC[74] := FALSE;
   PLI_HC[75] := FALSE;
   PLI_HC[76] := FALSE;
   PLI_HC[77] := FALSE;
   PLI_HC[78] := FALSE;
   PLI_HC[79] := FALSE;
   PLI_HC[80] := FALSE;
   PLI_HC[81] := FALSE;
   PLI_HC[82] := FALSE;
   PLI_HC[83] := FALSE;
   PLI_HC[84] := FALSE;
   PLI_HC[85] := FALSE;
   PLI_HC[86] := FALSE;
   PLI_HC[87] := FALSE;
   PLI_HC[88] := FALSE;
   PLI_HC[89] := FALSE;
   PLI_HC[90] := FALSE;
   PLI_HC[91] := FALSE;
   PLI_HC[92] := FALSE;
   PLI_HC[93] := FALSE;
   PLI_HC[94] := FALSE;
   PLI_HC[95] := FALSE;
   PLI_HC[96] := FALSE;
   PLI_HC[97] := FALSE;
   PLI_HC[98] := FALSE;
   PLI_HC[99] := FALSE;
   PLI_HC[100] := FALSE;
   PLI_HC[101] := FALSE;
   PLI_HC[102] := FALSE;
   PLI_HC[103] := FALSE;
   PLI_HC[104] := FALSE;
   PLI_HC[105] := FALSE;
   PLI_HC[106] := FALSE;
   PLI_HC[107] := FALSE;
   PLI_HC[108] := FALSE;
   PLI_HC[109] := FALSE;
   PLI_HC[110] := FALSE;
   PLI_HC[111] := FALSE;
   PLI_HC[112] := FALSE;
   PLI_HC[113] := FALSE;
   PLI_HC[114] := FALSE;
   PLI_HC[115] := FALSE;
   PLI_HC[116] := FALSE;
   PLI_HC[117] := FALSE;
   PLI_HC[118] := FALSE;
   PLI_HC[119] := FALSE;
   PLI_HC[120] := FALSE;
   PLI_HC[121] := FALSE;
   PLI_HC[122] := FALSE;
   PLI_HC[123] := FALSE;
   PLI_HC[124] := FALSE;
   PLI_HC[125] := FALSE;
   PLI_HC[126] := FALSE;
   PLI_HC[127] := FALSE;
   PLI_HC[128] := FALSE;
   PLI_HC[129] := FALSE;
   PLI_HC[130] := FALSE;
   PLI_HC[131] := FALSE;
   PLI_HC[132] := FALSE;
   PLI_HC[133] := FALSE;
   PLI_HC[134] := FALSE;
   PLI_HC[135] := FALSE;
   PLI_HC[136] := FALSE;
   PLI_HC[137] := FALSE;
   PLI_HC[138] := FALSE;
   PLI_HC[139] := FALSE;
   PLI_HC[140] := FALSE;
   PLI_HC[141] := FALSE;
   PLI_HC[142] := FALSE;
   PLI_HC[143] := FALSE;
   PLI_HC[144] := FALSE;
   PLI_HC[145] := FALSE;
   PLI_HC[146] := FALSE;
   PLI_HC[147] := FALSE;
   PLI_HC[148] := FALSE;
   PLI_HC[149] := FALSE;
   PLI_HC[150] := FALSE;
   PLI_SC[1] := FALSE;
   PLI_SC[2] := FALSE;
   PLI_SC[3] := FALSE;
   PLI_SC[4] := FALSE;
   PLI_SC[5] := FALSE;
   PLI_SC[6] := FALSE;
   PLI_SC[7] := FALSE;
   PLI_SC[8] := FALSE;
   PLI_SC[9] := FALSE;
   PLI_SC[10] := FALSE;
   PLI_SC[11] := FALSE;
   PLI_SC[12] := FALSE;
   PLI_SC[13] := FALSE;
   PLI_SC[14] := FALSE;
   PLI_SC[15] := FALSE;
   PLI_SC[16] := FALSE;
   PLI_SC[17] := FALSE;
   PLI_SC[18] := FALSE;
   PLI_SC[19] := FALSE;
   PLI_SC[20] := FALSE;
   PLI_SC[21] := FALSE;
   PLI_SC[22] := FALSE;
   PLI_SC[23] := FALSE;
   PLI_SC[24] := FALSE;
   PLI_SC[25] := FALSE;
   PLI_SC[26] := FALSE;
   PLI_SC[27] := FALSE;
   PLI_SC[28] := FALSE;
   PLI_SC[29] := FALSE;
   PLI_SC[30] := FALSE;
   PLI_SC[31] := FALSE;
   PLI_SC[32] := FALSE;
   PLI_SC[33] := FALSE;
   PLI_SC[34] := FALSE;
   PLI_SC[35] := FALSE;
   PLI_SC[36] := FALSE;
   PLI_SC[37] := FALSE;
   PLI_SC[38] := FALSE;
   PLI_SC[39] := FALSE;
   PLI_SC[40] := FALSE;
   PLI_SC[41] := FALSE;
   PLI_SC[42] := FALSE;
   PLI_SC[43] := FALSE;
   PLI_SC[44] := FALSE;
   PLI_SC[45] := FALSE;
   PLI_SC[46] := FALSE;
   PLI_SC[47] := FALSE;
   PLI_SC[48] := FALSE;
   PLI_SC[49] := FALSE;
   PLI_SC[50] := FALSE;
   PLI_SC[51] := FALSE;
   PLI_SC[52] := FALSE;
   PLI_SC[53] := FALSE;
   PLI_SC[54] := FALSE;
   PLI_SC[55] := FALSE;
   PLI_SC[56] := FALSE;
   PLI_SC[57] := FALSE;
   PLI_SC[58] := FALSE;
   PLI_SC[59] := FALSE;
   PLI_SC[60] := FALSE;
   PLI_SC[61] := FALSE;
   PLI_SC[62] := FALSE;
   PLI_SC[63] := FALSE;
   PLI_SC[64] := FALSE;
   PLI_SC[65] := FALSE;
   PLI_SC[66] := FALSE;
   PLI_SC[67] := FALSE;
   PLI_SC[68] := FALSE;
   PLI_SC[69] := FALSE;
   PLI_SC[70] := FALSE;
   PLI_SC[71] := FALSE;
   PLI_SC[72] := FALSE;
   PLI_SC[73] := FALSE;
   PLI_SC[74] := FALSE;
   PLI_SC[75] := FALSE;
   PLI_SC[76] := FALSE;
   PLI_SC[77] := FALSE;
   PLI_SC[78] := FALSE;
   PLI_SC[79] := FALSE;
   PLI_SC[80] := FALSE;
   PLI_SC[81] := FALSE;
   PLI_SC[82] := FALSE;
   PLI_SC[83] := FALSE;
   PLI_SC[84] := FALSE;
   PLI_SC[85] := FALSE;
   PLI_SC[86] := FALSE;
   PLI_SC[87] := FALSE;
   PLI_SC[88] := FALSE;
   PLI_SC[89] := FALSE;
   PLI_SC[90] := FALSE;
   PLI_SC[91] := FALSE;
   PLI_SC[92] := FALSE;
   PLI_SC[93] := FALSE;
   PLI_SC[94] := FALSE;
   PLI_SC[95] := FALSE;
   PLI_SC[96] := FALSE;
   PLI_SC[97] := FALSE;
   PLI_SC[98] := FALSE;
   PLI_SC[99] := FALSE;
   PLI_SC[100] := FALSE;
   PLI_SC[101] := FALSE;
   PLI_SC[102] := FALSE;
   PLI_SC[103] := FALSE;
   PLI_SC[104] := FALSE;
   PLI_SC[105] := FALSE;
   PLI_SC[106] := FALSE;
   PLI_SC[107] := FALSE;
   PLI_SC[108] := FALSE;
   PLI_SC[109] := FALSE;
   PLI_SC[110] := FALSE;
   PLI_SC[111] := FALSE;
   PLI_SC[112] := FALSE;
   PLI_SC[113] := FALSE;
   PLI_SC[114] := FALSE;
   PLI_SC[115] := FALSE;
   PLI_SC[116] := FALSE;
   PLI_SC[117] := FALSE;
   PLI_SC[118] := FALSE;
   PLI_SC[119] := FALSE;
   PLI_SC[120] := FALSE;
   PLI_SC[121] := FALSE;
   PLI_SC[122] := FALSE;
   PLI_SC[123] := FALSE;
   PLI_SC[124] := FALSE;
   PLI_SC[125] := FALSE;
   PLI_SC[126] := FALSE;
   PLI_SC[127] := FALSE;
   PLI_SC[128] := FALSE;
   PLI_SC[129] := FALSE;
   PLI_SC[130] := FALSE;
   PLI_SC[131] := FALSE;
   PLI_SC[132] := FALSE;
   PLI_SC[133] := FALSE;
   PLI_SC[134] := FALSE;
   PLI_SC[135] := FALSE;
   PLI_SC[136] := FALSE;
   PLI_SC[137] := FALSE;
   PLI_SC[138] := FALSE;
   PLI_SC[139] := FALSE;
   PLI_SC[140] := FALSE;
   PLI_SC[141] := FALSE;
   PLI_SC[142] := FALSE;
   PLI_SC[143] := FALSE;
   PLI_SC[144] := FALSE;
   PLI_SC[145] := FALSE;
   PLI_SC[146] := FALSE;
   PLI_SC[147] := FALSE;
   PLI_SC[148] := FALSE;
   PLI_SC[149] := FALSE;
   PLI_SC[150] := FALSE;
   PLI_EC[1] := FALSE;
   PLI_EC[2] := FALSE;
   PLI_EC[3] := FALSE;
   PLI_EC[4] := FALSE;
   PLI_EC[5] := FALSE;
   PLI_EC[6] := FALSE;
   PLI_EC[7] := FALSE;
   PLI_EC[8] := FALSE;
   PLI_EC[9] := FALSE;
   PLI_EC[10] := FALSE;
   PLI_EC[11] := FALSE;
   PLI_EC[12] := FALSE;
   PLI_EC[13] := FALSE;
   PLI_EC[14] := FALSE;
   PLI_EC[15] := FALSE;
   PLI_EC[16] := FALSE;
   PLI_EC[17] := FALSE;
   PLI_EC[18] := FALSE;
   PLI_EC[19] := FALSE;
   PLI_EC[20] := FALSE;
   PLI_EC[21] := FALSE;
   PLI_EC[22] := FALSE;
   PLI_EC[23] := FALSE;
   PLI_EC[24] := FALSE;
   PLI_EC[25] := FALSE;
   PLI_EC[26] := FALSE;
   PLI_EC[27] := FALSE;
   PLI_EC[28] := FALSE;
   PLI_EC[29] := FALSE;
   PLI_EC[30] := FALSE;
   PLI_EC[31] := FALSE;
   PLI_EC[32] := FALSE;
   PLI_EC[33] := FALSE;
   PLI_EC[34] := FALSE;
   PLI_EC[35] := FALSE;
   PLI_EC[36] := FALSE;
   PLI_EC[37] := FALSE;
   PLI_EC[38] := FALSE;
   PLI_EC[39] := FALSE;
   PLI_EC[40] := FALSE;
   PLI_EC[41] := FALSE;
   PLI_EC[42] := FALSE;
   PLI_EC[43] := FALSE;
   PLI_EC[44] := FALSE;
   PLI_EC[45] := FALSE;
   PLI_EC[46] := FALSE;
   PLI_EC[47] := FALSE;
   PLI_EC[48] := FALSE;
   PLI_EC[49] := FALSE;
   PLI_EC[50] := FALSE;
   PLI_EC[51] := FALSE;
   PLI_EC[52] := FALSE;
   PLI_EC[53] := FALSE;
   PLI_EC[54] := FALSE;
   PLI_EC[55] := FALSE;
   PLI_EC[56] := FALSE;
   PLI_EC[57] := FALSE;
   PLI_EC[58] := FALSE;
   PLI_EC[59] := FALSE;
   PLI_EC[60] := FALSE;
   PLI_EC[61] := FALSE;
   PLI_EC[62] := FALSE;
   PLI_EC[63] := FALSE;
   PLI_EC[64] := FALSE;
   PLI_EC[65] := FALSE;
   PLI_EC[66] := FALSE;
   PLI_EC[67] := FALSE;
   PLI_EC[68] := FALSE;
   PLI_EC[69] := FALSE;
   PLI_EC[70] := FALSE;
   PLI_EC[71] := FALSE;
   PLI_EC[72] := FALSE;
   PLI_EC[73] := FALSE;
   PLI_EC[74] := FALSE;
   PLI_EC[75] := FALSE;
   PLI_EC[76] := FALSE;
   PLI_EC[77] := FALSE;
   PLI_EC[78] := FALSE;
   PLI_EC[79] := FALSE;
   PLI_EC[80] := FALSE;
   PLI_EC[81] := FALSE;
   PLI_EC[82] := FALSE;
   PLI_EC[83] := FALSE;
   PLI_EC[84] := FALSE;
   PLI_EC[85] := FALSE;
   PLI_EC[86] := FALSE;
   PLI_EC[87] := FALSE;
   PLI_EC[88] := FALSE;
   PLI_EC[89] := FALSE;
   PLI_EC[90] := FALSE;
   PLI_EC[91] := FALSE;
   PLI_EC[92] := FALSE;
   PLI_EC[93] := FALSE;
   PLI_EC[94] := FALSE;
   PLI_EC[95] := FALSE;
   PLI_EC[96] := FALSE;
   PLI_EC[97] := FALSE;
   PLI_EC[98] := FALSE;
   PLI_EC[99] := FALSE;
   PLI_EC[100] := FALSE;
   PLI_EC[101] := FALSE;
   PLI_EC[102] := FALSE;
   PLI_EC[103] := FALSE;
   PLI_EC[104] := FALSE;
   PLI_EC[105] := FALSE;
   PLI_EC[106] := FALSE;
   PLI_EC[107] := FALSE;
   PLI_EC[108] := FALSE;
   PLI_EC[109] := FALSE;
   PLI_EC[110] := FALSE;
   PLI_EC[111] := FALSE;
   PLI_EC[112] := FALSE;
   PLI_EC[113] := FALSE;
   PLI_EC[114] := FALSE;
   PLI_EC[115] := FALSE;
   PLI_EC[116] := FALSE;
   PLI_EC[117] := FALSE;
   PLI_EC[118] := FALSE;
   PLI_EC[119] := FALSE;
   PLI_EC[120] := FALSE;
   PLI_EC[121] := FALSE;
   PLI_EC[122] := FALSE;
   PLI_EC[123] := FALSE;
   PLI_EC[124] := FALSE;
   PLI_EC[125] := FALSE;
   PLI_EC[126] := FALSE;
   PLI_EC[127] := FALSE;
   PLI_EC[128] := FALSE;
   PLI_EC[129] := FALSE;
   PLI_EC[130] := FALSE;
   PLI_EC[131] := FALSE;
   PLI_EC[132] := FALSE;
   PLI_EC[133] := FALSE;
   PLI_EC[134] := FALSE;
   PLI_EC[135] := FALSE;
   PLI_EC[136] := FALSE;
   PLI_EC[137] := FALSE;
   PLI_EC[138] := FALSE;
   PLI_EC[139] := FALSE;
   PLI_EC[140] := FALSE;
   PLI_EC[141] := FALSE;
   PLI_EC[142] := FALSE;
   PLI_EC[143] := FALSE;
